Yaskawa INFORM job: DEMO_ROOF_SIDE_0625_3PAINT_7.JBI

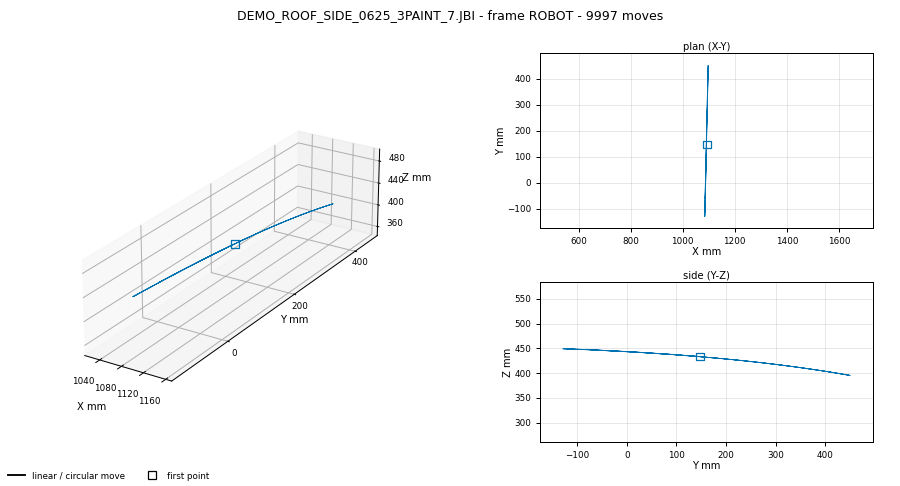
[picture p0: tool path of DEMO_ROOF_SIDE_0625_3PAINT_7.JBI in frame ROBOT, 9997 of 9997 moves have a stored position in this frame; points joined in program order, loops and branches not executed]
/JOB
//NAME DEMO_ROOF_SIDE_0625_3PAINT7
//POS
///NPOS 9997,0,0,0,0,0
///TOOL 0
///USER 0
///POSTYPE ROBOT
///RECTAN
///RCONF 1,0,0,0,0,0,0,0,0,0,0,0,0,0,0,0,0,0,0,0,0,0,0,0
C00000=1091.949,146.873,433.613,176.047,18.717,152.771
C00001=1091.943,146.623,433.633,176.045,18.716,152.771
C00002=1091.938,146.374,433.654,176.043,18.715,152.771
C00003=1091.932,146.126,433.675,176.040,18.714,152.771
C00004=1091.926,145.877,433.695,176.037,18.713,152.772
C00005=1091.921,145.628,433.716,176.034,18.712,152.772
C00006=1091.914,145.378,433.736,176.032,18.711,152.772
C00007=1091.909,145.129,433.757,176.029,18.710,152.772
C00008=1091.904,144.880,433.777,176.027,18.709,152.773
C00009=1091.899,144.631,433.798,176.024,18.708,152.773
C00010=1091.893,144.382,433.818,176.021,18.707,152.773
C00011=1091.886,144.106,433.841,176.018,18.706,152.773
C00012=1091.881,143.828,433.863,176.016,18.705,152.774
C00013=1091.874,143.552,433.886,176.013,18.704,152.774
C00014=1091.868,143.275,433.908,176.010,18.703,152.774
C00015=1091.862,143.026,433.929,176.007,18.702,152.775
C00016=1091.857,142.777,433.950,176.004,18.701,152.775
C00017=1091.851,142.527,433.970,176.002,18.700,152.775
C00018=1091.845,142.278,433.990,176.000,18.699,152.775
C00019=1091.839,142.029,434.010,175.997,18.698,152.776
C00020=1091.834,141.780,434.031,175.994,18.697,152.776
C00021=1091.829,141.531,434.051,175.991,18.696,152.776
C00022=1091.823,141.282,434.071,175.990,18.695,152.776
C00023=1091.818,141.033,434.092,175.987,18.694,152.777
C00024=1091.812,140.784,434.113,175.984,18.693,152.777
C00025=1091.806,140.535,434.133,175.981,18.692,152.777
C00026=1091.801,140.286,434.153,175.979,18.691,152.778
C00027=1091.795,140.036,434.173,175.977,18.690,152.778
C00028=1091.790,139.787,434.193,175.974,18.689,152.778
C00029=1091.784,139.538,434.213,175.971,18.688,152.778
C00030=1091.778,139.289,434.234,175.969,18.687,152.778
C00031=1091.772,139.040,434.254,175.967,18.686,152.779
C00032=1091.767,138.791,434.274,175.964,18.685,152.779
C00033=1091.761,138.542,434.293,175.961,18.683,152.779
C00034=1091.756,138.292,434.314,175.958,18.682,152.779
C00035=1091.750,138.044,434.334,175.957,18.682,152.780
C00036=1091.745,137.795,434.355,175.954,18.681,152.780
C00037=1091.739,137.546,434.375,175.951,18.679,152.780
C00038=1091.734,137.296,434.394,175.948,18.678,152.781
C00039=1091.728,137.047,434.414,175.946,18.678,152.781
C00040=1091.723,136.798,434.435,175.944,18.677,152.781
C00041=1091.717,136.549,434.455,175.941,18.676,152.781
C00042=1091.711,136.300,434.474,175.938,18.674,152.782
C00043=1091.706,136.051,434.495,175.936,18.674,152.782
C00044=1091.699,135.801,434.515,175.934,18.672,152.782
C00045=1091.694,135.552,434.536,175.931,18.671,152.782
C00046=1091.688,135.303,434.555,175.928,18.670,152.782
C00047=1091.682,135.054,434.575,175.926,18.669,152.783
C00048=1091.677,134.805,434.595,175.924,18.668,152.783
C00049=1091.671,134.555,434.615,175.921,18.667,152.783
C00050=1091.666,134.306,434.635,175.918,18.666,152.783
C00051=1091.661,134.058,434.655,175.916,18.665,152.784
C00052=1091.655,133.809,434.674,175.914,18.664,152.784
C00053=1091.650,133.559,434.694,175.911,18.663,152.784
C00054=1091.644,133.310,434.714,175.908,18.662,152.784
C00055=1091.638,133.061,434.734,175.906,18.661,152.785
C00056=1091.633,132.812,434.754,175.903,18.660,152.785
C00057=1091.627,132.563,434.773,175.901,18.658,152.785
C00058=1091.622,132.314,434.794,175.898,18.657,152.785
C00059=1091.616,132.064,434.813,175.896,18.657,152.785
C00060=1091.610,131.815,434.833,175.894,18.656,152.786
C00061=1091.604,131.566,434.853,175.891,18.655,152.786
C00062=1091.598,131.317,434.872,175.889,18.654,152.786
C00063=1091.593,131.068,434.893,175.886,18.652,152.786
C00064=1091.587,130.818,434.912,175.884,18.651,152.787
C00065=1091.581,130.570,434.932,175.881,18.650,152.787
C00066=1091.576,130.320,434.951,175.879,18.650,152.787
C00067=1091.570,130.071,434.971,175.876,18.648,152.787
C00068=1091.564,129.822,434.991,175.873,18.647,152.788
C00069=1091.559,129.573,435.011,175.871,18.646,152.788
C00070=1091.553,129.323,435.030,175.869,18.645,152.788
C00071=1091.547,129.075,435.050,175.866,18.644,152.788
C00072=1091.541,128.825,435.070,175.864,18.643,152.789
C00073=1091.536,128.576,435.089,175.862,18.642,152.789
C00074=1091.530,128.327,435.109,175.859,18.641,152.789
C00075=1091.524,128.050,435.131,175.856,18.640,152.789
C00076=1091.518,127.773,435.152,175.854,18.639,152.789
C00077=1091.511,127.496,435.174,175.851,18.637,152.790
C00078=1091.505,127.220,435.196,175.848,18.636,152.790
C00079=1091.499,126.970,435.215,175.845,18.635,152.790
C00080=1091.493,126.721,435.235,175.843,18.634,152.790
C00081=1091.488,126.472,435.254,175.841,18.633,152.791
C00082=1091.482,126.222,435.273,175.838,18.632,152.791
C00083=1091.477,125.974,435.294,175.836,18.630,152.791
C00084=1091.472,125.725,435.313,175.833,18.629,152.791
C00085=1091.466,125.475,435.332,175.831,18.629,152.792
C00086=1091.460,125.226,435.352,175.829,18.627,152.792
C00087=1091.454,124.977,435.371,175.826,18.626,152.792
C00088=1091.448,124.727,435.391,175.824,18.625,152.792
C00089=1091.442,124.479,435.411,175.821,18.624,152.792
C00090=1091.437,124.230,435.429,175.819,18.623,152.793
C00091=1091.432,123.980,435.449,175.817,18.622,152.793
C00092=1091.426,123.731,435.468,175.814,18.620,152.793
C00093=1091.420,123.482,435.488,175.811,18.619,152.793
C00094=1091.414,123.233,435.507,175.809,18.618,152.793
C00095=1091.409,122.983,435.526,175.807,18.617,152.794
C00096=1091.404,122.735,435.545,175.804,18.616,152.794
C00097=1091.398,122.485,435.564,175.802,18.615,152.794
C00098=1091.392,122.236,435.584,175.800,18.614,152.794
C00099=1091.386,121.987,435.604,175.797,18.613,152.794
C00100=1091.381,121.737,435.623,175.795,18.611,152.795
C00101=1091.376,121.488,435.642,175.793,18.611,152.795
C00102=1091.370,121.239,435.662,175.790,18.609,152.795
C00103=1091.365,120.990,435.681,175.787,18.608,152.795
C00104=1091.359,120.741,435.701,175.786,18.607,152.795
C00105=1091.353,120.491,435.720,175.783,18.606,152.796
C00106=1091.348,120.243,435.739,175.780,18.605,152.796
C00107=1091.342,119.993,435.758,175.778,18.603,152.796
C00108=1091.337,119.744,435.777,175.776,18.602,152.796
C00109=1091.331,119.494,435.797,175.773,18.601,152.796
C00110=1091.326,119.246,435.816,175.771,18.600,152.797
C00111=1091.320,118.996,435.835,175.769,18.599,152.797
C00112=1091.314,118.747,435.853,175.766,18.598,152.797
C00113=1091.309,118.498,435.872,175.764,18.596,152.797
C00114=1091.303,118.249,435.892,175.762,18.595,152.797
C00115=1091.297,117.999,435.911,175.759,18.594,152.797
C00116=1091.292,117.750,435.930,175.757,18.593,152.798
C00117=1091.287,117.501,435.949,175.755,18.592,152.798
C00118=1091.281,117.252,435.968,175.752,18.590,152.798
C00119=1091.275,117.002,435.987,175.750,18.589,152.798
C00120=1091.270,116.754,436.006,175.748,18.588,152.798
C00121=1091.264,116.504,436.026,175.745,18.587,152.798
C00122=1091.259,116.255,436.045,175.743,18.585,152.799
C00123=1091.254,116.006,436.064,175.741,18.585,152.799
C00124=1091.248,115.757,436.083,175.738,18.583,152.799
C00125=1091.242,115.507,436.102,175.736,18.581,152.799
C00126=1091.237,115.258,436.121,175.734,18.581,152.799
C00127=1091.231,115.009,436.140,175.731,18.579,152.799
C00128=1091.226,114.760,436.160,175.729,18.578,152.800
C00129=1091.220,114.511,436.178,175.726,18.577,152.800
C00130=1091.214,114.262,436.197,175.724,18.575,152.800
C00131=1091.209,114.012,436.216,175.722,18.574,152.800
C00132=1091.204,113.763,436.234,175.720,18.573,152.800
C00133=1091.198,113.514,436.254,175.717,18.572,152.801
C00134=1091.192,113.264,436.272,175.715,18.571,152.801
C00135=1091.187,113.016,436.291,175.713,18.570,152.801
C00136=1091.181,112.766,436.310,175.710,18.568,152.801
C00137=1091.175,112.517,436.330,175.708,18.567,152.801
C00138=1091.170,112.268,436.347,175.706,18.566,152.801
C00139=1091.164,111.990,436.369,175.703,18.565,152.802
C00140=1091.157,111.714,436.390,175.701,18.564,152.802
C00141=1091.151,111.437,436.411,175.698,18.562,152.802
C00142=1091.145,111.160,436.431,175.695,18.561,152.802
C00143=1091.139,110.911,436.451,175.693,18.559,152.802
C00144=1091.133,110.661,436.468,175.690,18.558,152.802
C00145=1091.128,110.413,436.487,175.689,18.557,152.803
C00146=1091.122,110.163,436.507,175.686,18.555,152.803
C00147=1091.116,109.915,436.525,175.684,18.555,152.803
C00148=1091.111,109.665,436.543,175.682,18.553,152.803
C00149=1091.104,109.416,436.562,175.679,18.552,152.803
C00150=1091.099,109.167,436.581,175.677,18.551,152.804
C00151=1091.094,108.917,436.599,175.675,18.550,152.804
C00152=1091.087,108.668,436.618,175.672,18.548,152.804
C00153=1091.082,108.419,436.637,175.670,18.547,152.804
C00154=1091.076,108.169,436.655,175.668,18.546,152.804
C00155=1091.071,107.920,436.674,175.665,18.545,152.804
C00156=1091.065,107.671,436.693,175.663,18.544,152.805
C00157=1091.059,107.421,436.711,175.661,18.542,152.805
C00158=1091.054,107.173,436.730,175.658,18.540,152.805
C00159=1091.048,106.923,436.748,175.657,18.540,152.805
C00160=1091.043,106.674,436.767,175.654,18.538,152.805
C00161=1091.037,106.425,436.785,175.652,18.537,152.805
C00162=1091.031,106.175,436.804,175.650,18.536,152.806
C00163=1091.026,105.926,436.823,175.647,18.534,152.806
C00164=1091.020,105.677,436.841,175.645,18.533,152.806
C00165=1091.015,105.428,436.859,175.643,18.532,152.806
C00166=1091.008,105.179,436.878,175.640,18.531,152.806
C00167=1091.004,104.929,436.896,175.639,18.530,152.806
C00168=1090.997,104.680,436.915,175.636,18.528,152.806
C00169=1090.993,104.431,436.933,175.634,18.527,152.806
C00170=1090.986,104.182,436.952,175.632,18.526,152.807
C00171=1090.981,103.932,436.970,175.629,18.524,152.807
C00172=1090.975,103.683,436.989,175.627,18.523,152.807
C00173=1090.970,103.434,437.007,175.625,18.522,152.807
C00174=1090.964,103.185,437.025,175.622,18.521,152.807
C00175=1090.959,102.935,437.044,175.621,18.519,152.807
C00176=1090.952,102.686,437.062,175.618,18.518,152.808
C00177=1090.948,102.437,437.080,175.616,18.517,152.808
C00178=1090.942,102.187,437.098,175.614,18.515,152.808
C00179=1090.936,101.938,437.117,175.611,18.514,152.808
C00180=1090.930,101.689,437.135,175.609,18.513,152.808
C00181=1090.925,101.440,437.154,175.607,18.511,152.808
C00182=1090.919,101.190,437.172,175.604,18.510,152.808
C00183=1090.914,100.941,437.191,175.603,18.509,152.808
C00184=1090.908,100.692,437.209,175.600,18.507,152.809
C00185=1090.902,100.443,437.226,175.598,18.507,152.809
C00186=1090.897,100.193,437.246,175.596,18.505,152.809
C00187=1090.891,99.944,437.263,175.593,18.503,152.809
C00188=1090.885,99.694,437.281,175.592,18.502,152.809
C00189=1090.880,99.446,437.300,175.589,18.501,152.809
C00190=1090.874,99.196,437.318,175.587,18.500,152.810
C00191=1090.868,98.947,437.335,175.585,18.499,152.810
C00192=1090.863,98.697,437.355,175.582,18.497,152.810
C00193=1090.857,98.448,437.372,175.581,18.496,152.810
C00194=1090.851,98.199,437.390,175.578,18.494,152.810
C00195=1090.845,97.950,437.408,175.577,18.493,152.810
C00196=1090.840,97.700,437.427,175.574,18.492,152.810
C00197=1090.834,97.451,437.445,175.571,18.491,152.811
C00198=1090.828,97.201,437.462,175.570,18.489,152.811
C00199=1090.823,96.953,437.481,175.567,18.488,152.811
C00200=1090.817,96.703,437.499,175.565,18.487,152.811
C00201=1090.811,96.454,437.517,175.563,18.485,152.811
C00202=1090.806,96.205,437.534,175.560,18.484,152.811
C00203=1090.800,95.928,437.555,175.559,18.483,152.811
C00204=1090.793,95.650,437.575,175.556,18.481,152.811
C00205=1090.787,95.374,437.595,175.554,18.479,152.811
C00206=1090.781,95.098,437.615,175.551,18.478,152.812
C00207=1090.775,94.849,437.633,175.549,18.477,152.812
C00208=1090.770,94.599,437.651,175.547,18.476,152.812
C00209=1090.764,94.350,437.669,175.544,18.474,152.812
C00210=1090.759,94.100,437.687,175.543,18.473,152.812
C00211=1090.752,93.851,437.705,175.540,18.471,152.812
C00212=1090.747,93.602,437.722,175.538,18.470,152.812
C00213=1090.742,93.353,437.741,175.536,18.469,152.812
C00214=1090.736,93.103,437.759,175.534,18.467,152.813
C00215=1090.730,92.854,437.777,175.532,18.466,152.813
C00216=1090.725,92.605,437.794,175.529,18.464,152.813
C00217=1090.719,92.355,437.813,175.527,18.463,152.813
C00218=1090.714,92.106,437.830,175.525,18.462,152.813
C00219=1090.708,91.857,437.848,175.523,18.460,152.813
C00220=1090.702,91.607,437.866,175.521,18.459,152.813
C00221=1090.697,91.358,437.883,175.519,18.458,152.813
C00222=1090.692,91.109,437.901,175.517,18.456,152.814
C00223=1090.686,90.859,437.919,175.514,18.455,152.814
C00224=1090.680,90.610,437.937,175.512,18.453,152.814
C00225=1090.674,90.360,437.955,175.510,18.452,152.814
C00226=1090.669,90.111,437.972,175.508,18.451,152.814
C00227=1090.663,89.862,437.990,175.506,18.450,152.814
C00228=1090.657,89.613,438.008,175.504,18.448,152.814
C00229=1090.651,89.363,438.025,175.502,18.447,152.814
C00230=1090.646,89.114,438.043,175.499,18.445,152.814
C00231=1090.640,88.865,438.061,175.497,18.444,152.815
C00232=1090.634,88.616,438.079,175.495,18.443,152.815
C00233=1090.629,88.367,438.096,175.493,18.441,152.815
C00234=1090.623,88.117,438.114,175.491,18.440,152.815
C00235=1090.617,87.868,438.132,175.489,18.438,152.815
C00236=1090.612,87.619,438.149,175.487,18.437,152.815
C00237=1090.605,87.369,438.167,175.485,18.436,152.815
C00238=1090.600,87.120,438.185,175.482,18.434,152.815
C00239=1090.594,86.871,438.202,175.480,18.433,152.815
C00240=1090.589,86.621,438.219,175.478,18.431,152.816
C00241=1090.583,86.372,438.237,175.476,18.430,152.816
C00242=1090.578,86.123,438.255,175.474,18.429,152.816
C00243=1090.571,85.873,438.273,175.472,18.427,152.816
C00244=1090.566,85.624,438.290,175.470,18.426,152.816
C00245=1090.560,85.375,438.308,175.468,18.425,152.816
C00246=1090.554,85.126,438.325,175.466,18.423,152.816
C00247=1090.548,84.876,438.342,175.463,18.421,152.816
C00248=1090.543,84.627,438.359,175.461,18.420,152.816
C00249=1090.537,84.378,438.377,175.459,18.419,152.816
C00250=1090.532,84.129,438.395,175.457,18.418,152.817
C00251=1090.526,83.879,438.412,175.455,18.416,152.817
C00252=1090.520,83.629,438.429,175.453,18.414,152.817
C00253=1090.515,83.380,438.447,175.451,18.413,152.817
C00254=1090.509,83.131,438.464,175.449,18.412,152.817
C00255=1090.503,82.881,438.482,175.447,18.410,152.817
C00256=1090.498,82.632,438.499,175.444,18.409,152.817
C00257=1090.493,82.383,438.517,175.443,18.408,152.817
C00258=1090.487,82.134,438.534,175.440,18.406,152.817
C00259=1090.482,81.884,438.551,175.439,18.404,152.817
C00260=1090.475,81.634,438.569,175.436,18.403,152.817
C00261=1090.469,81.385,438.586,175.435,18.402,152.817
C00262=1090.464,81.136,438.604,175.432,18.400,152.818
C00263=1090.459,80.887,438.621,175.430,18.399,152.818
C00264=1090.453,80.638,438.638,175.428,18.397,152.818
C00265=1090.448,80.389,438.656,175.427,18.396,152.818
C00266=1090.442,80.138,438.673,175.424,18.394,152.818
C00267=1090.436,79.862,438.692,175.422,18.393,152.818
C00268=1090.429,79.585,438.711,175.419,18.391,152.818
C00269=1090.423,79.308,438.730,175.418,18.390,152.818
C00270=1090.416,79.032,438.749,175.415,18.388,152.818
C00271=1090.411,78.782,438.767,175.413,18.386,152.818
C00272=1090.406,78.533,438.784,175.411,18.385,152.818
C00273=1090.400,78.284,438.801,175.409,18.383,152.818
C00274=1090.395,78.034,438.818,175.407,18.382,152.819
C00275=1090.389,77.785,438.835,175.405,18.381,152.819
C00276=1090.383,77.536,438.853,175.403,18.379,152.819
C00277=1090.377,77.286,438.870,175.401,18.377,152.819
C00278=1090.371,77.037,438.887,175.399,18.376,152.819
C00279=1090.366,76.788,438.904,175.397,18.375,152.819
C00280=1090.360,76.539,438.921,175.394,18.373,152.819
C00281=1090.355,76.289,438.938,175.392,18.372,152.819
C00282=1090.348,76.039,438.955,175.390,18.370,152.819
C00283=1090.343,75.790,438.972,175.388,18.369,152.819
C00284=1090.338,75.541,438.990,175.386,18.367,152.819
C00285=1090.332,75.291,439.006,175.384,18.366,152.820
C00286=1090.326,75.042,439.024,175.382,18.364,152.820
C00287=1090.321,74.793,439.041,175.380,18.363,152.820
C00288=1090.315,74.544,439.057,175.378,18.362,152.820
C00289=1090.309,74.294,439.074,175.377,18.360,152.820
C00290=1090.303,74.045,439.092,175.374,18.358,152.820
C00291=1090.297,73.795,439.109,175.372,18.357,152.820
C00292=1090.292,73.546,439.125,175.370,18.356,152.820
C00293=1090.286,73.297,439.142,175.368,18.354,152.820
C00294=1090.281,73.047,439.159,175.366,18.353,152.820
C00295=1090.275,72.798,439.177,175.364,18.351,152.820
C00296=1090.269,72.549,439.193,175.362,18.349,152.820
C00297=1090.264,72.299,439.210,175.360,18.348,152.820
C00298=1090.258,72.050,439.227,175.358,18.347,152.820
C00299=1090.252,71.801,439.244,175.357,18.345,152.820
C00300=1090.247,71.551,439.261,175.354,18.344,152.821
C00301=1090.240,71.302,439.278,175.352,18.342,152.821
C00302=1090.235,71.052,439.295,175.350,18.340,152.821
C00303=1090.230,70.802,439.312,175.348,18.339,152.821
C00304=1090.224,70.554,439.329,175.346,18.338,152.821
C00305=1090.219,70.304,439.345,175.345,18.336,152.821
C00306=1090.213,70.055,439.362,175.342,18.335,152.821
C00307=1090.207,69.806,439.379,175.340,18.333,152.821
C00308=1090.201,69.556,439.395,175.338,18.331,152.821
C00309=1090.196,69.307,439.412,175.337,18.330,152.821
C00310=1090.190,69.058,439.429,175.334,18.329,152.821
C00311=1090.184,68.808,439.446,175.333,18.327,152.821
C00312=1090.178,68.559,439.462,175.330,18.326,152.821
C00313=1090.173,68.309,439.479,175.328,18.325,152.821
C00314=1090.167,68.060,439.496,175.326,18.322,152.821
C00315=1090.162,67.811,439.513,175.325,18.321,152.821
C00316=1090.156,67.561,439.529,175.322,18.319,152.821
C00317=1090.151,67.312,439.546,175.321,18.318,152.822
C00318=1090.145,67.062,439.562,175.318,18.317,152.822
C00319=1090.138,66.814,439.579,175.317,18.315,152.822
C00320=1090.133,66.564,439.596,175.314,18.313,152.822
C00321=1090.127,66.315,439.613,175.313,18.312,152.822
C00322=1090.122,66.065,439.629,175.310,18.310,152.822
C00323=1090.116,65.816,439.646,175.309,18.309,152.822
C00324=1090.111,65.566,439.662,175.307,18.307,152.822
C00325=1090.105,65.317,439.679,175.305,18.306,152.822
C00326=1090.099,65.068,439.696,175.303,18.304,152.822
C00327=1090.093,64.818,439.713,175.301,18.303,152.822
C00328=1090.088,64.569,439.729,175.298,18.301,152.822
C00329=1090.082,64.319,439.746,175.297,18.300,152.822
C00330=1090.076,64.070,439.762,175.295,18.298,152.822
C00331=1090.069,63.793,439.781,175.293,18.297,152.822
C00332=1090.063,63.516,439.799,175.291,18.295,152.822
C00333=1090.057,63.239,439.816,175.288,18.293,152.823
C00334=1090.050,62.963,439.836,175.286,18.291,152.823
C00335=1090.044,62.713,439.852,175.284,18.290,152.823
C00336=1090.038,62.464,439.868,175.282,18.289,152.823
C00337=1090.032,62.215,439.884,175.280,18.287,152.823
C00338=1090.027,61.965,439.901,175.278,18.285,152.823
C00339=1090.021,61.716,439.918,175.277,18.284,152.823
C00340=1090.015,61.466,439.934,175.274,18.282,152.823
C00341=1090.009,61.217,439.950,175.272,18.281,152.823
C00342=1090.004,60.967,439.967,175.271,18.280,152.823
C00343=1089.998,60.718,439.983,175.268,18.278,152.823
C00344=1089.992,60.468,439.999,175.267,18.276,152.823
C00345=1089.986,60.219,440.016,175.265,18.275,152.823
C00346=1089.980,59.970,440.032,175.263,18.273,152.823
C00347=1089.975,59.721,440.048,175.261,18.272,152.823
C00348=1089.969,59.471,440.065,175.259,18.271,152.823
C00349=1089.964,59.222,440.081,175.257,18.269,152.823
C00350=1089.958,58.973,440.097,175.255,18.268,152.823
C00351=1089.952,58.723,440.113,175.253,18.265,152.823
C00352=1089.946,58.473,440.129,175.251,18.264,152.824
C00353=1089.941,58.224,440.146,175.249,18.262,152.824
C00354=1089.935,57.974,440.162,175.247,18.261,152.824
C00355=1089.929,57.725,440.178,175.245,18.259,152.824
C00356=1089.923,57.476,440.195,175.243,18.258,152.824
C00357=1089.917,57.226,440.211,175.242,18.256,152.824
C00358=1089.911,56.977,440.227,175.240,18.255,152.824
C00359=1089.905,56.728,440.243,175.238,18.253,152.824
C00360=1089.901,56.478,440.259,175.236,18.252,152.824
C00361=1089.895,56.229,440.275,175.234,18.250,152.824
C00362=1089.889,55.979,440.292,175.232,18.249,152.824
C00363=1089.883,55.730,440.308,175.230,18.247,152.824
C00364=1089.877,55.481,440.324,175.228,18.245,152.824
C00365=1089.871,55.231,440.340,175.226,18.244,152.824
C00366=1089.865,54.981,440.356,175.224,18.242,152.824
C00367=1089.859,54.732,440.372,175.223,18.241,152.824
C00368=1089.855,54.483,440.389,175.221,18.240,152.824
C00369=1089.849,54.234,440.405,175.219,18.237,152.824
C00370=1089.843,53.984,440.420,175.217,18.236,152.824
C00371=1089.837,53.734,440.437,175.215,18.234,152.824
C00372=1089.831,53.485,440.453,175.213,18.233,152.824
C00373=1089.825,53.236,440.469,175.211,18.231,152.824
C00374=1089.820,52.986,440.484,175.210,18.230,152.824
C00375=1089.814,52.737,440.501,175.207,18.228,152.824
C00376=1089.808,52.488,440.517,175.206,18.226,152.824
C00377=1089.802,52.238,440.533,175.204,18.225,152.824
C00378=1089.797,51.988,440.549,175.202,18.223,152.824
C00379=1089.791,51.740,440.565,175.200,18.222,152.824
C00380=1089.786,51.490,440.581,175.198,18.220,152.825
C00381=1089.781,51.240,440.597,175.196,18.219,152.824
C00382=1089.775,50.991,440.613,175.194,18.216,152.824
C00383=1089.769,50.741,440.630,175.193,18.215,152.825
C00384=1089.764,50.492,440.645,175.190,18.213,152.825
C00385=1089.758,50.243,440.661,175.189,18.212,152.824
C00386=1089.752,49.993,440.677,175.187,18.211,152.825
C00387=1089.746,49.744,440.693,175.185,18.209,152.825
C00388=1089.741,49.495,440.709,175.184,18.207,152.825
C00389=1089.735,49.245,440.724,175.181,18.205,152.825
C00390=1089.729,48.996,440.740,175.180,18.204,152.825
C00391=1089.724,48.746,440.756,175.178,18.202,152.825
C00392=1089.718,48.497,440.772,175.176,18.201,152.825
C00393=1089.712,48.248,440.788,175.174,18.199,152.825
C00394=1089.707,47.998,440.804,175.172,18.197,152.825
C00395=1089.700,47.721,440.821,175.170,18.195,152.825
C00396=1089.694,47.443,440.839,175.168,18.194,152.825
C00397=1089.688,47.167,440.856,175.166,18.192,152.825
C00398=1089.682,46.890,440.874,175.164,18.190,152.825
C00399=1089.676,46.640,440.889,175.162,18.189,152.825
C00400=1089.670,46.391,440.906,175.160,18.186,152.825
C00401=1089.665,46.142,440.921,175.159,18.185,152.825
C00402=1089.659,45.892,440.937,175.157,18.184,152.825
C00403=1089.653,45.642,440.953,175.155,18.182,152.825
C00404=1089.648,45.394,440.969,175.153,18.180,152.825
C00405=1089.642,45.144,440.984,175.151,18.178,152.825
C00406=1089.636,44.894,441.000,175.149,18.177,152.825
C00407=1089.631,44.645,441.016,175.147,18.175,152.825
C00408=1089.625,44.396,441.032,175.146,18.173,152.825
C00409=1089.620,44.146,441.047,175.144,18.172,152.825
C00410=1089.615,43.896,441.063,175.142,18.170,152.825
C00411=1089.609,43.647,441.079,175.141,18.169,152.825
C00412=1089.603,43.397,441.094,175.138,18.166,152.825
C00413=1089.598,43.148,441.110,175.137,18.165,152.825
C00414=1089.591,42.899,441.125,175.135,18.164,152.825
C00415=1089.586,42.649,441.141,175.133,18.162,152.825
C00416=1089.580,42.400,441.157,175.132,18.160,152.825
C00417=1089.575,42.150,441.172,175.129,18.159,152.825
C00418=1089.569,41.901,441.188,175.128,18.157,152.825
C00419=1089.562,41.651,441.203,175.126,18.155,152.825
C00420=1089.557,41.402,441.219,175.124,18.154,152.825
C00421=1089.551,41.153,441.235,175.122,18.152,152.825
C00422=1089.546,40.903,441.250,175.120,18.150,152.825
C00423=1089.540,40.654,441.265,175.119,18.149,152.825
C00424=1089.534,40.404,441.281,175.116,18.147,152.825
C00425=1089.529,40.155,441.296,175.115,18.145,152.825
C00426=1089.523,39.905,441.312,175.114,18.144,152.825
C00427=1089.517,39.655,441.327,175.111,18.142,152.825
C00428=1089.512,39.407,441.343,175.110,18.141,152.825
C00429=1089.506,39.157,441.358,175.107,18.139,152.825
C00430=1089.500,38.907,441.374,175.106,18.137,152.825
C00431=1089.495,38.658,441.388,175.104,18.136,152.825
C00432=1089.489,38.409,441.405,175.102,18.134,152.825
C00433=1089.484,38.159,441.420,175.101,18.132,152.825
C00434=1089.478,37.909,441.435,175.099,18.130,152.825
C00435=1089.472,37.660,441.450,175.097,18.129,152.825
C00436=1089.466,37.411,441.466,175.095,18.128,152.825
C00437=1089.461,37.161,441.482,175.093,18.125,152.825
C00438=1089.454,36.911,441.497,175.092,18.124,152.825
C00439=1089.449,36.662,441.512,175.090,18.123,152.825
C00440=1089.443,36.412,441.527,175.088,18.121,152.825
C00441=1089.437,36.164,441.543,175.087,18.119,152.825
C00442=1089.431,35.914,441.558,175.084,18.117,152.825
C00443=1089.425,35.664,441.573,175.083,18.116,152.825
C00444=1089.420,35.415,441.588,175.081,18.114,152.825
C00445=1089.414,35.165,441.603,175.079,18.112,152.825
C00446=1089.408,34.915,441.619,175.077,18.111,152.825
C00447=1089.402,34.667,441.634,175.075,18.109,152.825
C00448=1089.397,34.417,441.650,175.074,18.108,152.825
C00449=1089.391,34.168,441.664,175.072,18.106,152.825
C00450=1089.385,33.918,441.680,175.070,18.104,152.825
C00451=1089.380,33.669,441.695,175.068,18.103,152.825
C00452=1089.374,33.419,441.710,175.067,18.101,152.825
C00453=1089.368,33.169,441.725,175.065,18.099,152.825
C00454=1089.362,32.920,441.740,175.063,18.098,152.825
C00455=1089.357,32.670,441.756,175.061,18.096,152.825
C00456=1089.351,32.421,441.770,175.060,18.094,152.825
C00457=1089.345,32.171,441.786,175.058,18.093,152.825
C00458=1089.339,31.922,441.800,175.056,18.091,152.825
C00459=1089.333,31.646,441.818,175.055,18.089,152.825
C00460=1089.326,31.368,441.835,175.052,18.088,152.825
C00461=1089.320,31.091,441.852,175.050,18.085,152.825
C00462=1089.314,30.814,441.868,175.048,18.084,152.825
C00463=1089.309,30.565,441.883,175.046,18.082,152.825
C00464=1089.302,30.315,441.898,175.045,18.080,152.825
C00465=1089.297,30.066,441.913,175.043,18.079,152.825
C00466=1089.291,29.816,441.928,175.041,18.077,152.825
C00467=1089.286,29.567,441.943,175.040,18.075,152.825
C00468=1089.279,29.317,441.958,175.038,18.074,152.825
C00469=1089.274,29.068,441.973,175.036,18.072,152.825
C00470=1089.268,28.819,441.988,175.035,18.070,152.825
C00471=1089.263,28.569,442.004,175.032,18.068,152.825
C00472=1089.256,28.320,442.018,175.031,18.067,152.825
C00473=1089.251,28.070,442.034,175.029,18.065,152.825
C00474=1089.245,27.820,442.048,175.027,18.063,152.825
C00475=1089.240,27.571,442.062,175.026,18.062,152.825
C00476=1089.234,27.321,442.078,175.024,18.060,152.825
C00477=1089.228,27.072,442.093,175.022,18.059,152.825
C00478=1089.222,26.823,442.108,175.020,18.057,152.825
C00479=1089.217,26.573,442.123,175.019,18.055,152.825
C00480=1089.210,26.324,442.138,175.017,18.053,152.825
C00481=1089.204,26.075,442.152,175.015,18.052,152.825
C00482=1089.199,25.825,442.168,175.014,18.051,152.825
C00483=1089.193,25.575,442.182,175.011,18.049,152.825
C00484=1089.187,25.325,442.197,175.010,18.047,152.825
C00485=1089.182,25.076,442.212,175.008,18.045,152.825
C00486=1089.176,24.827,442.227,175.006,18.043,152.825
C00487=1089.170,24.578,442.241,175.005,18.042,152.825
C00488=1089.164,24.327,442.256,175.003,18.040,152.825
C00489=1089.159,24.078,442.271,175.001,18.039,152.825
C00490=1089.152,23.828,442.286,175.000,18.037,152.825
C00491=1089.147,23.579,442.301,174.998,18.035,152.825
C00492=1089.141,23.329,442.316,174.996,18.033,152.825
C00493=1089.135,23.080,442.330,174.995,18.032,152.825
C00494=1089.130,22.831,442.345,174.992,18.030,152.825
C00495=1089.124,22.581,442.360,174.991,18.029,152.825
C00496=1089.118,22.332,442.374,174.990,18.027,152.825
C00497=1089.112,22.082,442.389,174.987,18.025,152.825
C00498=1089.107,21.832,442.404,174.986,18.023,152.825
C00499=1089.101,21.584,442.418,174.985,18.022,152.825
C00500=1089.095,21.334,442.433,174.982,18.020,152.825
C00501=1089.089,21.084,442.447,174.981,18.019,152.825
C00502=1089.084,20.834,442.463,174.979,18.017,152.825
C00503=1089.078,20.585,442.477,174.977,18.015,152.825
C00504=1089.073,20.336,442.491,174.976,18.013,152.825
C00505=1089.066,20.086,442.506,174.974,18.012,152.825
C00506=1089.061,19.837,442.521,174.972,18.010,152.825
C00507=1089.055,19.587,442.535,174.971,18.008,152.825
C00508=1089.049,19.338,442.550,174.969,18.007,152.825
C00509=1089.043,19.089,442.565,174.967,18.005,152.825
C00510=1089.037,18.838,442.579,174.965,18.003,152.825
C00511=1089.032,18.589,442.593,174.964,18.002,152.825
C00512=1089.026,18.339,442.608,174.962,18.000,152.825
C00513=1089.020,18.090,442.623,174.960,17.998,152.825
C00514=1089.015,17.841,442.637,174.959,17.997,152.824
C00515=1089.009,17.591,442.652,174.957,17.994,152.824
C00516=1089.003,17.342,442.666,174.955,17.993,152.825
C00517=1088.997,17.091,442.680,174.954,17.992,152.825
C00518=1088.991,16.842,442.695,174.951,17.990,152.825
C00519=1088.986,16.593,442.710,174.950,17.988,152.824
C00520=1088.980,16.343,442.724,174.949,17.987,152.824
C00521=1088.974,16.094,442.739,174.946,17.984,152.824
C00522=1088.969,15.844,442.753,174.945,17.983,152.824
C00523=1088.962,15.569,442.769,174.944,17.981,152.824
C00524=1088.956,15.293,442.785,174.941,17.979,152.824
C00525=1088.949,15.017,442.800,174.939,17.977,152.824
C00526=1088.943,14.742,442.817,174.938,17.975,152.824
C00527=1088.937,14.492,442.831,174.936,17.974,152.824
C00528=1088.931,14.243,442.845,174.934,17.972,152.824
C00529=1088.925,13.993,442.860,174.933,17.971,152.824
C00530=1088.919,13.744,442.874,174.931,17.969,152.824
C00531=1088.914,13.494,442.888,174.929,17.967,152.824
C00532=1088.907,13.245,442.903,174.928,17.965,152.824
C00533=1088.902,12.995,442.917,174.926,17.964,152.824
C00534=1088.896,12.746,442.932,174.924,17.962,152.824
C00535=1088.890,12.496,442.946,174.922,17.961,152.824
C00536=1088.885,12.246,442.960,174.921,17.959,152.824
C00537=1088.879,11.997,442.974,174.919,17.957,152.824
C00538=1088.873,11.747,442.988,174.917,17.955,152.824
C00539=1088.867,11.498,443.003,174.916,17.954,152.824
C00540=1088.862,11.249,443.017,174.915,17.952,152.824
C00541=1088.854,10.999,443.031,174.912,17.951,152.824
C00542=1088.849,10.750,443.045,174.911,17.949,152.824
C00543=1088.843,10.500,443.059,174.909,17.948,152.824
C00544=1088.837,10.250,443.074,174.907,17.945,152.824
C00545=1088.832,10.001,443.088,174.906,17.944,152.824
C00546=1088.826,9.751,443.102,174.904,17.942,152.824
C00547=1088.820,9.502,443.117,174.902,17.940,152.824
C00548=1088.814,9.252,443.130,174.900,17.939,152.824
C00549=1088.809,9.002,443.144,174.899,17.938,152.824
C00550=1088.803,8.754,443.159,174.898,17.936,152.824
C00551=1088.796,8.504,443.173,174.895,17.934,152.824
C00552=1088.791,8.254,443.186,174.894,17.932,152.824
C00553=1088.785,8.005,443.201,174.893,17.931,152.824
C00554=1088.779,7.755,443.215,174.890,17.929,152.824
C00555=1088.773,7.505,443.229,174.889,17.927,152.824
C00556=1088.768,7.256,443.244,174.888,17.925,152.824
C00557=1088.762,7.007,443.257,174.886,17.924,152.824
C00558=1088.757,6.757,443.271,174.884,17.922,152.824
C00559=1088.750,6.507,443.285,174.882,17.921,152.824
C00560=1088.744,6.258,443.300,174.881,17.919,152.824
C00561=1088.739,6.009,443.313,174.879,17.917,152.824
C00562=1088.733,5.759,443.327,174.877,17.915,152.824
C00563=1088.727,5.509,443.342,174.876,17.914,152.824
C00564=1088.722,5.259,443.355,174.875,17.912,152.824
C00565=1088.715,5.011,443.369,174.872,17.910,152.824
C00566=1088.710,4.761,443.383,174.871,17.909,152.824
C00567=1088.704,4.511,443.397,174.870,17.907,152.824
C00568=1088.698,4.261,443.411,174.867,17.905,152.824
C00569=1088.693,4.012,443.425,174.866,17.904,152.824
C00570=1088.687,3.763,443.440,174.864,17.902,152.824
C00571=1088.681,3.513,443.453,174.863,17.901,152.824
C00572=1088.675,3.264,443.467,174.861,17.899,152.824
C00573=1088.669,3.013,443.481,174.859,17.897,152.824
C00574=1088.664,2.764,443.495,174.858,17.895,152.823
C00575=1088.658,2.514,443.509,174.856,17.893,152.823
C00576=1088.652,2.265,443.522,174.854,17.892,152.823
C00577=1088.646,2.016,443.537,174.853,17.890,152.823
C00578=1088.641,1.767,443.551,174.852,17.889,152.823
C00579=1088.634,1.516,443.565,174.849,17.886,152.823
C00580=1088.629,1.267,443.579,174.848,17.885,152.823
C00581=1088.623,1.017,443.592,174.847,17.883,152.823
C00582=1088.617,0.768,443.606,174.845,17.882,152.823
C00583=1088.612,0.518,443.620,174.843,17.880,152.823
C00584=1088.606,0.269,443.634,174.842,17.878,152.823
C00585=1088.601,0.019,443.647,174.840,17.877,152.823
C00586=1088.595,-0.230,443.661,174.838,17.875,152.823
C00587=1088.589,-0.504,443.676,174.836,17.873,152.823
C00588=1088.582,-0.778,443.691,174.835,17.871,152.823
C00589=1088.575,-1.052,443.706,174.833,17.869,152.823
C00590=1088.569,-1.325,443.721,174.832,17.867,152.823
C00591=1088.564,-1.575,443.735,174.829,17.865,152.823
C00592=1088.558,-1.825,443.749,174.828,17.864,152.823
C00593=1088.552,-2.074,443.762,174.827,17.862,152.823
C00594=1088.547,-2.323,443.776,174.824,17.860,152.823
C00595=1088.541,-2.573,443.790,174.823,17.859,152.823
C00596=1088.536,-2.822,443.804,174.821,17.857,152.823
C00597=1088.529,-3.072,443.817,174.820,17.856,152.823
C00598=1088.524,-3.321,443.831,174.818,17.854,152.823
C00599=1088.518,-3.571,443.845,174.816,17.852,152.823
C00600=1088.512,-3.821,443.859,174.815,17.851,152.823
C00601=1088.506,-4.070,443.872,174.814,17.849,152.823
C00602=1088.500,-4.320,443.886,174.811,17.847,152.823
C00603=1088.494,-4.569,443.900,174.810,17.845,152.823
C00604=1088.488,-4.819,443.913,174.809,17.844,152.823
C00605=1088.483,-5.068,443.927,174.807,17.842,152.823
C00606=1088.477,-5.317,443.940,174.805,17.841,152.823
C00607=1088.471,-5.567,443.954,174.803,17.839,152.823
C00608=1088.465,-5.817,443.966,174.802,17.837,152.823
C00609=1088.459,-6.067,443.981,174.800,17.836,152.823
C00610=1088.453,-6.316,443.994,174.798,17.834,152.823
C00611=1088.447,-6.566,444.008,174.797,17.832,152.823
C00612=1088.441,-6.815,444.021,174.796,17.831,152.822
C00613=1088.436,-7.065,444.035,174.794,17.829,152.822
C00614=1088.429,-7.314,444.048,174.793,17.827,152.822
C00615=1088.424,-7.564,444.061,174.790,17.826,152.823
C00616=1088.418,-7.814,444.075,174.789,17.824,152.822
C00617=1088.413,-8.063,444.088,174.787,17.823,152.822
C00618=1088.406,-8.312,444.102,174.786,17.821,152.822
C00619=1088.401,-8.562,444.116,174.784,17.819,152.822
C00620=1088.395,-8.811,444.129,174.782,17.817,152.822
C00621=1088.390,-9.061,444.142,174.781,17.816,152.822
C00622=1088.383,-9.311,444.156,174.780,17.814,152.822
C00623=1088.377,-9.561,444.169,174.777,17.812,152.822
C00624=1088.371,-9.810,444.183,174.776,17.811,152.822
C00625=1088.366,-10.060,444.196,174.775,17.809,152.822
C00626=1088.360,-10.310,444.209,174.773,17.808,152.822
C00627=1088.353,-10.559,444.222,174.771,17.806,152.822
C00628=1088.348,-10.809,444.236,174.769,17.804,152.822
C00629=1088.342,-11.058,444.249,174.768,17.803,152.822
C00630=1088.337,-11.308,444.263,174.767,17.801,152.822
C00631=1088.330,-11.557,444.276,174.765,17.799,152.822
C00632=1088.325,-11.807,444.289,174.763,17.797,152.822
C00633=1088.319,-12.057,444.302,174.762,17.796,152.822
C00634=1088.314,-12.306,444.316,174.760,17.794,152.822
C00635=1088.307,-12.556,444.329,174.759,17.793,152.822
C00636=1088.301,-12.805,444.342,174.757,17.790,152.822
C00637=1088.296,-13.055,444.356,174.755,17.789,152.822
C00638=1088.290,-13.304,444.369,174.754,17.787,152.822
C00639=1088.285,-13.554,444.382,174.752,17.786,152.822
C00640=1088.278,-13.804,444.396,174.751,17.785,152.822
C00641=1088.272,-14.054,444.408,174.749,17.783,152.822
C00642=1088.268,-14.302,444.422,174.747,17.781,152.822
C00643=1088.261,-14.552,444.435,174.746,17.779,152.822
C00644=1088.256,-14.802,444.448,174.745,17.778,152.822
C00645=1088.250,-15.051,444.461,174.742,17.776,152.822
C00646=1088.244,-15.300,444.475,174.741,17.774,152.822
C00647=1088.239,-15.551,444.488,174.740,17.773,152.822
C00648=1088.232,-15.800,444.501,174.738,17.771,152.822
C00649=1088.226,-16.050,444.514,174.737,17.770,152.822
C00650=1088.220,-16.299,444.527,174.734,17.768,152.822
C00651=1088.214,-16.572,444.541,174.733,17.766,152.822
C00652=1088.207,-16.843,444.555,174.732,17.765,152.822
C00653=1088.201,-17.115,444.569,174.729,17.762,152.822
C00654=1088.195,-17.387,444.584,174.728,17.761,152.822
C00655=1088.189,-17.637,444.598,174.727,17.759,152.822
C00656=1088.183,-17.887,444.610,174.724,17.757,152.822
C00657=1088.176,-18.136,444.623,174.723,17.756,152.821
C00658=1088.171,-18.386,444.637,174.722,17.754,152.821
C00659=1088.165,-18.635,444.650,174.720,17.753,152.822
C00660=1088.159,-18.885,444.662,174.719,17.751,152.822
C00661=1088.153,-19.134,444.676,174.716,17.749,152.822
C00662=1088.148,-19.384,444.688,174.715,17.748,152.821
C00663=1088.142,-19.633,444.702,174.714,17.746,152.821
C00664=1088.136,-19.883,444.714,174.712,17.745,152.821
C00665=1088.130,-20.132,444.728,174.711,17.743,152.821
C00666=1088.124,-20.382,444.740,174.708,17.741,152.821
C00667=1088.118,-20.632,444.753,174.707,17.740,152.821
C00668=1088.112,-20.881,444.766,174.706,17.738,152.821
C00669=1088.107,-21.132,444.779,174.704,17.737,152.821
C00670=1088.101,-21.381,444.792,174.703,17.735,152.821
C00671=1088.095,-21.631,444.805,174.701,17.733,152.821
C00672=1088.088,-21.880,444.818,174.699,17.731,152.821
C00673=1088.083,-22.129,444.830,174.698,17.730,152.821
C00674=1088.077,-22.379,444.843,174.696,17.729,152.821
C00675=1088.072,-22.629,444.857,174.695,17.727,152.821
C00676=1088.066,-22.879,444.869,174.693,17.725,152.821
C00677=1088.060,-23.128,444.883,174.691,17.723,152.821
C00678=1088.054,-23.378,444.895,174.690,17.722,152.821
C00679=1088.048,-23.628,444.908,174.688,17.720,152.821
C00680=1088.042,-23.876,444.921,174.687,17.719,152.821
C00681=1088.036,-24.126,444.933,174.686,17.717,152.821
C00682=1088.031,-24.376,444.946,174.683,17.715,152.821
C00683=1088.025,-24.625,444.960,174.682,17.714,152.821
C00684=1088.019,-24.875,444.972,174.680,17.712,152.821
C00685=1088.013,-25.125,444.985,174.679,17.711,152.821
C00686=1088.007,-25.374,444.998,174.678,17.709,152.821
C00687=1088.002,-25.624,445.010,174.675,17.707,152.821
C00688=1087.996,-25.874,445.023,174.674,17.705,152.821
C00689=1087.990,-26.123,445.035,174.673,17.704,152.821
C00690=1087.984,-26.373,445.049,174.671,17.703,152.821
C00691=1087.978,-26.623,445.062,174.670,17.701,152.821
C00692=1087.973,-26.872,445.074,174.668,17.700,152.821
C00693=1087.967,-27.121,445.087,174.666,17.697,152.821
C00694=1087.961,-27.371,445.100,174.665,17.696,152.821
C00695=1087.955,-27.621,445.112,174.663,17.694,152.821
C00696=1087.949,-27.871,445.125,174.662,17.693,152.821
C00697=1087.943,-28.120,445.138,174.660,17.692,152.821
C00698=1087.937,-28.370,445.151,174.659,17.690,152.821
C00699=1087.931,-28.619,445.162,174.657,17.688,152.821
C00700=1087.925,-28.869,445.175,174.655,17.686,152.821
C00701=1087.919,-29.119,445.187,174.654,17.685,152.821
C00702=1087.913,-29.368,445.201,174.652,17.684,152.821
C00703=1087.907,-29.618,445.213,174.651,17.682,152.821
C00704=1087.901,-29.868,445.226,174.649,17.681,152.821
C00705=1087.896,-30.117,445.238,174.648,17.679,152.821
C00706=1087.890,-30.367,445.250,174.646,17.677,152.821
C00707=1087.884,-30.616,445.264,174.644,17.676,152.821
C00708=1087.878,-30.866,445.276,174.643,17.674,152.821
C00709=1087.872,-31.116,445.289,174.641,17.673,152.821
C00710=1087.867,-31.365,445.301,174.640,17.671,152.821
C00711=1087.860,-31.615,445.313,174.638,17.670,152.821
C00712=1087.854,-31.865,445.325,174.636,17.668,152.821
C00713=1087.848,-32.114,445.338,174.635,17.666,152.821
C00714=1087.842,-32.363,445.351,174.633,17.665,152.821
C00715=1087.836,-32.635,445.364,174.632,17.663,152.821
C00716=1087.830,-32.906,445.378,174.630,17.661,152.821
C00717=1087.823,-33.177,445.392,174.628,17.660,152.821
C00718=1087.817,-33.448,445.406,174.627,17.658,152.821
C00719=1087.811,-33.697,445.418,174.625,17.657,152.821
C00720=1087.805,-33.947,445.430,174.624,17.655,152.821
C00721=1087.799,-34.197,445.443,174.622,17.653,152.821
C00722=1087.793,-34.447,445.455,174.620,17.651,152.821
C00723=1087.787,-34.696,445.467,174.619,17.650,152.821
C00724=1087.782,-34.946,445.480,174.617,17.649,152.821
C00725=1087.776,-35.196,445.492,174.616,17.647,152.821
C00726=1087.770,-35.445,445.504,174.615,17.646,152.821
C00727=1087.764,-35.695,445.517,174.613,17.644,152.821
C00728=1087.759,-35.945,445.529,174.611,17.642,152.821
C00729=1087.752,-36.194,445.541,174.609,17.641,152.821
C00730=1087.747,-36.443,445.554,174.608,17.639,152.821
C00731=1087.741,-36.693,445.566,174.607,17.638,152.821
C00732=1087.735,-36.943,445.579,174.605,17.636,152.821
C00733=1087.729,-37.192,445.591,174.604,17.635,152.821
C00734=1087.724,-37.442,445.603,174.602,17.633,152.821
C00735=1087.717,-37.692,445.615,174.601,17.632,152.821
C00736=1087.712,-37.941,445.628,174.599,17.630,152.821
C00737=1087.706,-38.191,445.640,174.597,17.628,152.821
C00738=1087.700,-38.441,445.653,174.596,17.627,152.821
C00739=1087.694,-38.690,445.665,174.594,17.625,152.821
C00740=1087.688,-38.940,445.677,174.593,17.624,152.821
C00741=1087.682,-39.189,445.689,174.591,17.622,152.820
C00742=1087.676,-39.439,445.702,174.590,17.621,152.821
C00743=1087.670,-39.689,445.713,174.588,17.620,152.821
C00744=1087.664,-39.939,445.725,174.586,17.618,152.821
C00745=1087.658,-40.189,445.738,174.585,17.616,152.821
C00746=1087.652,-40.437,445.749,174.583,17.615,152.821
C00747=1087.647,-40.687,445.762,174.582,17.613,152.821
C00748=1087.641,-40.937,445.775,174.580,17.612,152.821
C00749=1087.634,-41.187,445.787,174.579,17.611,152.821
C00750=1087.629,-41.436,445.799,174.577,17.609,152.821
C00751=1087.623,-41.686,445.811,174.576,17.607,152.821
C00752=1087.616,-41.936,445.823,174.574,17.606,152.821
C00753=1087.611,-42.185,445.835,174.572,17.604,152.821
C00754=1087.604,-42.435,445.847,174.571,17.603,152.821
C00755=1087.599,-42.685,445.859,174.569,17.601,152.821
C00756=1087.593,-42.934,445.871,174.568,17.600,152.821
C00757=1087.587,-43.184,445.883,174.566,17.598,152.821
C00758=1087.581,-43.434,445.895,174.565,17.597,152.821
C00759=1087.576,-43.683,445.907,174.563,17.596,152.821
C00760=1087.569,-43.933,445.919,174.562,17.594,152.821
C00761=1087.563,-44.183,445.932,174.561,17.593,152.821
C00762=1087.557,-44.432,445.943,174.558,17.591,152.821
C00763=1087.551,-44.682,445.955,174.557,17.589,152.821
C00764=1087.546,-44.931,445.968,174.555,17.588,152.821
C00765=1087.540,-45.181,445.979,174.554,17.586,152.821
C00766=1087.534,-45.431,445.992,174.552,17.585,152.821
C00767=1087.528,-45.680,446.003,174.551,17.584,152.821
C00768=1087.522,-45.930,446.015,174.550,17.582,152.821
C00769=1087.517,-46.179,446.028,174.548,17.581,152.821
C00770=1087.510,-46.429,446.039,174.547,17.579,152.821
C00771=1087.504,-46.679,446.051,174.545,17.578,152.821
C00772=1087.498,-46.928,446.063,174.543,17.577,152.821
C00773=1087.492,-47.178,446.076,174.541,17.575,152.821
C00774=1087.487,-47.427,446.086,174.540,17.573,152.821
C00775=1087.481,-47.677,446.099,174.538,17.572,152.821
C00776=1087.475,-47.927,446.112,174.537,17.570,152.821
C00777=1087.469,-48.177,446.122,174.535,17.569,152.821
C00778=1087.463,-48.427,446.135,174.534,17.567,152.821
C00779=1087.456,-48.698,446.148,174.532,17.566,152.821
C00780=1087.450,-48.969,446.161,174.531,17.564,152.821
C00781=1087.444,-49.240,446.174,174.529,17.562,152.821
C00782=1087.437,-49.512,446.186,174.527,17.561,152.821
C00783=1087.432,-49.762,446.198,174.526,17.560,152.821
C00784=1087.425,-50.011,446.210,174.524,17.558,152.821
C00785=1087.420,-50.262,446.222,174.523,17.556,152.821
C00786=1087.414,-50.511,446.233,174.521,17.555,152.821
C00787=1087.408,-50.761,446.245,174.520,17.554,152.821
C00788=1087.402,-51.010,446.257,174.518,17.553,152.821
C00789=1087.396,-51.260,446.269,174.516,17.551,152.821
C00790=1087.390,-51.510,446.281,174.515,17.550,152.821
C00791=1087.384,-51.759,446.292,174.513,17.548,152.821
C00792=1087.378,-52.009,446.304,174.512,17.546,152.821
C00793=1087.372,-52.258,446.316,174.510,17.545,152.821
C00794=1087.366,-52.508,446.328,174.509,17.544,152.821
C00795=1087.359,-52.758,446.339,174.507,17.543,152.821
C00796=1087.354,-53.007,446.351,174.506,17.541,152.821
C00797=1087.348,-53.257,446.362,174.504,17.540,152.821
C00798=1087.342,-53.506,446.374,174.503,17.538,152.821
C00799=1087.335,-53.756,446.385,174.501,17.537,152.821
C00800=1087.329,-54.006,446.398,174.500,17.536,152.821
C00801=1087.324,-54.256,446.409,174.498,17.534,152.821
C00802=1087.317,-54.505,446.421,174.497,17.533,152.821
C00803=1087.311,-54.755,446.431,174.495,17.531,152.821
C00804=1087.305,-55.005,446.444,174.494,17.530,152.821
C00805=1087.300,-55.254,446.455,174.492,17.529,152.821
C00806=1087.293,-55.504,446.467,174.491,17.528,152.821
C00807=1087.288,-55.754,446.478,174.489,17.526,152.821
C00808=1087.281,-56.003,446.490,174.487,17.525,152.822
C00809=1087.275,-56.253,446.502,174.485,17.523,152.822
C00810=1087.269,-56.502,446.513,174.484,17.522,152.822
C00811=1087.263,-56.753,446.525,174.482,17.520,152.822
C00812=1087.257,-57.002,446.537,174.481,17.519,152.822
C00813=1087.251,-57.252,446.548,174.479,17.518,152.822
C00814=1087.245,-57.501,446.559,174.478,17.517,152.822
C00815=1087.238,-57.751,446.571,174.476,17.515,152.822
C00816=1087.233,-58.001,446.582,174.475,17.513,152.822
C00817=1087.227,-58.250,446.594,174.473,17.512,152.822
C00818=1087.221,-58.500,446.605,174.472,17.511,152.822
C00819=1087.214,-58.749,446.617,174.470,17.510,152.822
C00820=1087.209,-58.999,446.628,174.469,17.508,152.822
C00821=1087.203,-59.249,446.640,174.467,17.507,152.822
C00822=1087.197,-59.498,446.651,174.466,17.505,152.822
C00823=1087.191,-59.748,446.662,174.464,17.504,152.822
C00824=1087.185,-59.998,446.673,174.463,17.503,152.822
C00825=1087.179,-60.248,446.686,174.461,17.502,152.822
C00826=1087.173,-60.497,446.697,174.460,17.500,152.822
C00827=1087.167,-60.747,446.708,174.458,17.499,152.822
C00828=1087.161,-60.996,446.720,174.457,17.497,152.822
C00829=1087.155,-61.246,446.730,174.455,17.496,152.822
C00830=1087.150,-61.496,446.742,174.454,17.495,152.822
C00831=1087.144,-61.745,446.754,174.452,17.494,152.822
C00832=1087.137,-61.995,446.765,174.451,17.492,152.822
C00833=1087.131,-62.245,446.776,174.449,17.491,152.822
C00834=1087.125,-62.494,446.788,174.448,17.489,152.822
C00835=1087.119,-62.744,446.799,174.446,17.488,152.822
C00836=1087.113,-62.994,446.811,174.445,17.487,152.822
C00837=1087.108,-63.244,446.822,174.443,17.486,152.822
C00838=1087.102,-63.493,446.833,174.442,17.484,152.822
C00839=1087.095,-63.743,446.844,174.440,17.483,152.823
C00840=1087.090,-63.992,446.855,174.439,17.481,152.822
C00841=1087.083,-64.243,446.867,174.437,17.480,152.823
C00842=1087.078,-64.492,446.879,174.436,17.479,152.823
C00843=1087.071,-64.765,446.890,174.433,17.477,152.823
C00844=1087.065,-65.037,446.903,174.432,17.476,152.823
C00845=1087.058,-65.310,446.916,174.430,17.474,152.823
C00846=1087.052,-65.583,446.927,174.429,17.473,152.823
C00847=1087.046,-65.833,446.938,174.427,17.472,152.823
C00848=1087.040,-66.082,446.951,174.426,17.470,152.823
C00849=1087.034,-66.332,446.961,174.424,17.469,152.823
C00850=1087.028,-66.582,446.973,174.423,17.468,152.823
C00851=1087.022,-66.832,446.984,174.421,17.466,152.823
C00852=1087.017,-67.081,446.994,174.419,17.465,152.823
C00853=1087.010,-67.331,447.006,174.418,17.464,152.823
C00854=1087.004,-67.580,447.017,174.416,17.463,152.823
C00855=1086.998,-67.830,447.028,174.415,17.461,152.823
C00856=1086.992,-68.080,447.039,174.413,17.460,152.823
C00857=1086.987,-68.330,447.051,174.412,17.458,152.823
C00858=1086.981,-68.580,447.062,174.410,17.457,152.823
C00859=1086.975,-68.829,447.073,174.409,17.456,152.823
C00860=1086.969,-69.079,447.084,174.407,17.455,152.823
C00861=1086.963,-69.329,447.095,174.406,17.453,152.823
C00862=1086.957,-69.578,447.107,174.404,17.452,152.823
C00863=1086.951,-69.827,447.118,174.403,17.451,152.824
C00864=1086.945,-70.077,447.128,174.401,17.449,152.824
C00865=1086.939,-70.327,447.140,174.399,17.448,152.824
C00866=1086.933,-70.576,447.151,174.398,17.447,152.824
C00867=1086.928,-70.826,447.161,174.396,17.446,152.824
C00868=1086.922,-71.076,447.173,174.395,17.444,152.824
C00869=1086.916,-71.326,447.184,174.393,17.443,152.824
C00870=1086.911,-71.575,447.195,174.392,17.442,152.824
C00871=1086.904,-71.826,447.206,174.390,17.440,152.824
C00872=1086.899,-72.075,447.217,174.389,17.439,152.824
C00873=1086.893,-72.325,447.228,174.387,17.438,152.824
C00874=1086.887,-72.574,447.239,174.386,17.437,152.824
C00875=1086.881,-72.824,447.250,174.384,17.435,152.824
C00876=1086.875,-73.074,447.261,174.383,17.434,152.824
C00877=1086.869,-73.323,447.272,174.381,17.433,152.824
C00878=1086.863,-73.573,447.283,174.380,17.431,152.824
C00879=1086.857,-73.823,447.294,174.378,17.430,152.824
C00880=1086.851,-74.072,447.305,174.377,17.429,152.824
C00881=1086.846,-74.322,447.316,174.375,17.428,152.824
C00882=1086.840,-74.571,447.327,174.373,17.426,152.824
C00883=1086.834,-74.822,447.338,174.373,17.425,152.824
C00884=1086.828,-75.071,447.349,174.371,17.424,152.824
C00885=1086.822,-75.321,447.360,174.370,17.423,152.825
C00886=1086.815,-75.570,447.370,174.368,17.422,152.825
C00887=1086.809,-75.820,447.381,174.366,17.421,152.825
C00888=1086.804,-76.069,447.392,174.365,17.420,152.825
C00889=1086.797,-76.320,447.403,174.363,17.418,152.825
C00890=1086.791,-76.569,447.414,174.362,17.417,152.825
C00891=1086.786,-76.819,447.425,174.360,17.416,152.825
C00892=1086.780,-77.068,447.436,174.359,17.415,152.825
C00893=1086.773,-77.319,447.446,174.357,17.413,152.825
C00894=1086.767,-77.568,447.457,174.355,17.412,152.825
C00895=1086.762,-77.818,447.468,174.354,17.411,152.825
C00896=1086.756,-78.067,447.478,174.352,17.410,152.825
C00897=1086.750,-78.317,447.490,174.351,17.408,152.825
C00898=1086.744,-78.567,447.501,174.349,17.407,152.825
C00899=1086.737,-78.816,447.511,174.348,17.406,152.826
C00900=1086.732,-79.065,447.522,174.346,17.405,152.826
C00901=1086.726,-79.316,447.532,174.345,17.404,152.826
C00902=1086.720,-79.566,447.543,174.344,17.403,152.826
C00903=1086.714,-79.815,447.554,174.342,17.402,152.826
C00904=1086.708,-80.064,447.564,174.341,17.400,152.826
C00905=1086.701,-80.315,447.576,174.339,17.399,152.826
C00906=1086.696,-80.564,447.586,174.337,17.398,152.826
C00907=1086.689,-80.839,447.598,174.336,17.397,152.826
C00908=1086.682,-81.114,447.609,174.334,17.396,152.826
C00909=1086.675,-81.389,447.621,174.332,17.395,152.826
C00910=1086.669,-81.664,447.633,174.330,17.393,152.826
C00911=1086.663,-81.914,447.644,174.329,17.392,152.826
C00912=1086.656,-82.164,447.654,174.328,17.391,152.826
C00913=1086.650,-82.413,447.665,174.326,17.390,152.827
C00914=1086.645,-82.663,447.675,174.324,17.389,152.827
C00915=1086.638,-82.913,447.686,174.323,17.388,152.827
C00916=1086.632,-83.163,447.697,174.321,17.386,152.827
C00917=1086.626,-83.412,447.708,174.320,17.385,152.827
C00918=1086.620,-83.662,447.717,174.318,17.384,152.827
C00919=1086.614,-83.911,447.728,174.316,17.383,152.827
C00920=1086.607,-84.161,447.739,174.315,17.382,152.827
C00921=1086.602,-84.411,447.750,174.313,17.381,152.827
C00922=1086.596,-84.661,447.760,174.312,17.380,152.827
C00923=1086.590,-84.910,447.770,174.311,17.379,152.827
C00924=1086.583,-85.160,447.781,174.309,17.378,152.827
C00925=1086.577,-85.410,447.791,174.308,17.377,152.828
C00926=1086.571,-85.659,447.802,174.306,17.376,152.828
C00927=1086.566,-85.909,447.813,174.304,17.375,152.828
C00928=1086.559,-86.158,447.823,174.303,17.373,152.828
C00929=1086.553,-86.409,447.833,174.301,17.372,152.828
C00930=1086.547,-86.658,447.844,174.299,17.371,152.828
C00931=1086.541,-86.908,447.855,174.298,17.370,152.828
C00932=1086.535,-87.158,447.865,174.297,17.369,152.828
C00933=1086.529,-87.407,447.875,174.296,17.368,152.828
C00934=1086.523,-87.658,447.886,174.294,17.367,152.828
C00935=1086.516,-87.907,447.896,174.292,17.366,152.828
C00936=1086.511,-88.156,447.907,174.291,17.365,152.829
C00937=1086.505,-88.406,447.917,174.289,17.364,152.829
C00938=1086.499,-88.656,447.927,174.287,17.363,152.829
C00939=1086.493,-88.905,447.938,174.286,17.362,152.829
C00940=1086.486,-89.156,447.948,174.285,17.361,152.829
C00941=1086.481,-89.405,447.959,174.283,17.360,152.829
C00942=1086.474,-89.655,447.968,174.282,17.359,152.829
C00943=1086.469,-89.904,447.979,174.280,17.357,152.829
C00944=1086.462,-90.154,447.990,174.279,17.356,152.829
C00945=1086.457,-90.404,448.000,174.277,17.355,152.829
C00946=1086.451,-90.653,448.011,174.275,17.354,152.830
C00947=1086.445,-90.903,448.020,174.274,17.353,152.830
C00948=1086.439,-91.153,448.031,174.273,17.353,152.830
C00949=1086.432,-91.403,448.041,174.271,17.351,152.830
C00950=1086.427,-91.652,448.052,174.269,17.350,152.830
C00951=1086.420,-91.902,448.061,174.268,17.349,152.830
C00952=1086.415,-92.152,448.072,174.266,17.348,152.830
C00953=1086.409,-92.402,448.082,174.264,17.347,152.830
C00954=1086.403,-92.651,448.093,174.263,17.346,152.830
C00955=1086.397,-92.901,448.102,174.261,17.345,152.830
C00956=1086.391,-93.150,448.113,174.260,17.344,152.831
C00957=1086.384,-93.401,448.123,174.259,17.343,152.831
C00958=1086.378,-93.650,448.134,174.257,17.342,152.831
C00959=1086.372,-93.900,448.144,174.255,17.341,152.831
C00960=1086.366,-94.150,448.154,174.254,17.340,152.831
C00961=1086.360,-94.399,448.164,174.252,17.339,152.831
C00962=1086.355,-94.649,448.175,174.250,17.338,152.831
C00963=1086.348,-94.899,448.184,174.250,17.337,152.831
C00964=1086.343,-95.148,448.195,174.248,17.336,152.831
C00965=1086.336,-95.398,448.205,174.246,17.335,152.831
C00966=1086.331,-95.647,448.216,174.245,17.334,152.832
C00967=1086.325,-95.897,448.225,174.243,17.333,152.832
C00968=1086.319,-96.147,448.236,174.242,17.332,152.832
C00969=1086.313,-96.397,448.246,174.241,17.331,152.832
C00970=1086.307,-96.647,448.256,174.239,17.330,152.832
C00971=1086.300,-96.924,448.267,174.237,17.329,152.832
C00972=1086.293,-97.201,448.279,174.236,17.328,152.832
C00973=1086.287,-97.478,448.290,174.234,17.327,152.832
C00974=1086.280,-97.755,448.301,174.232,17.326,152.832
C00975=1086.274,-98.005,448.311,174.231,17.325,152.833
C00976=1086.268,-98.255,448.322,174.229,17.324,152.833
C00977=1086.262,-98.504,448.331,174.227,17.323,152.833
C00978=1086.256,-98.754,448.341,174.226,17.322,152.833
C00979=1086.250,-99.004,448.352,174.224,17.321,152.833
C00980=1086.243,-99.254,448.362,174.223,17.320,152.833
C00981=1086.237,-99.504,448.371,174.222,17.319,152.833
C00982=1086.231,-99.754,448.382,174.220,17.319,152.833
C00983=1086.225,-100.003,448.392,174.218,17.318,152.834
C00984=1086.219,-100.253,448.401,174.216,17.316,152.834
C00985=1086.213,-100.502,448.411,174.215,17.315,152.834
C00986=1086.207,-100.752,448.422,174.214,17.315,152.834
C00987=1086.201,-101.002,448.431,174.212,17.314,152.834
C00988=1086.195,-101.251,448.441,174.211,17.313,152.834
C00989=1086.189,-101.502,448.452,174.209,17.312,152.834
C00990=1086.183,-101.751,448.461,174.207,17.311,152.834
C00991=1086.176,-102.001,448.472,174.206,17.311,152.835
C00992=1086.170,-102.250,448.481,174.205,17.309,152.835
C00993=1086.165,-102.500,448.491,174.203,17.308,152.835
C00994=1086.159,-102.750,448.501,174.201,17.307,152.835
C00995=1086.152,-102.999,448.511,174.200,17.306,152.835
C00996=1086.146,-103.249,448.521,174.199,17.306,152.835
C00997=1086.141,-103.499,448.531,174.197,17.305,152.835
C00998=1086.134,-103.749,448.540,174.195,17.304,152.835
C00999=1086.128,-103.998,448.551,174.194,17.303,152.836
C01000=1086.122,-104.248,448.560,174.192,17.302,152.836
C01001=1086.116,-104.498,448.570,174.191,17.302,152.836
C01002=1086.110,-104.748,448.580,174.189,17.301,152.836
C01003=1086.104,-104.998,448.590,174.188,17.300,152.836
C01004=1086.098,-105.247,448.600,174.186,17.299,152.836
C01005=1086.092,-105.497,448.610,174.184,17.298,152.836
C01006=1086.086,-105.747,448.620,174.183,17.298,152.837
C01007=1086.080,-105.997,448.629,174.181,17.297,152.837
C01008=1086.074,-106.246,448.639,174.180,17.295,152.837
C01009=1086.067,-106.496,448.649,174.178,17.294,152.837
C01010=1086.062,-106.746,448.659,174.177,17.293,152.837
C01011=1086.055,-106.996,448.669,174.175,17.293,152.837
C01012=1086.049,-107.245,448.678,174.174,17.292,152.837
C01013=1086.043,-107.495,448.688,174.172,17.291,152.837
C01014=1086.037,-107.745,448.697,174.170,17.290,152.838
C01015=1086.030,-107.994,448.708,174.169,17.290,152.838
C01016=1086.024,-108.244,448.717,174.168,17.289,152.838
C01017=1086.019,-108.494,448.727,174.166,17.288,152.838
C01018=1086.013,-108.744,448.737,174.164,17.287,152.838
C01019=1086.007,-108.994,448.747,174.163,17.286,152.838
C01020=1086.000,-109.243,448.756,174.162,17.286,152.838
C01021=1085.994,-109.493,448.766,174.160,17.285,152.839
C01022=1085.988,-109.743,448.775,174.158,17.284,152.839
C01023=1085.982,-109.993,448.785,174.156,17.283,152.839
C01024=1085.975,-110.242,448.795,174.155,17.283,152.839
C01025=1085.969,-110.492,448.805,174.154,17.282,152.839
C01026=1085.964,-110.741,448.814,174.152,17.281,152.839
C01027=1085.957,-110.991,448.823,174.150,17.280,152.840
C01028=1085.951,-111.240,448.833,174.149,17.280,152.840
C01029=1085.945,-111.490,448.843,174.148,17.279,152.840
C01030=1085.940,-111.740,448.853,174.146,17.278,152.840
C01031=1085.934,-111.990,448.862,174.144,17.277,152.840
C01032=1085.927,-112.240,448.872,174.143,17.276,152.840
C01033=1085.921,-112.490,448.881,174.141,17.276,152.841
C01034=1085.915,-112.740,448.891,174.140,17.275,152.841
C01035=1085.908,-113.012,448.902,174.138,17.274,152.841
C01036=1085.902,-113.284,448.911,174.136,17.273,152.841
C01037=1085.895,-113.557,448.922,174.134,17.272,152.841
C01038=1085.888,-113.830,448.932,174.133,17.272,152.841
C01039=1085.882,-114.079,448.942,174.132,17.271,152.841
C01040=1085.876,-114.328,448.951,174.130,17.270,152.842
C01041=1085.870,-114.578,448.961,174.128,17.269,152.842
C01042=1085.864,-114.828,448.970,174.126,17.268,152.842
C01043=1085.858,-115.078,448.980,174.125,17.268,152.842
C01044=1085.852,-115.328,448.989,174.124,17.267,152.842
C01045=1085.846,-115.577,448.999,174.122,17.266,152.842
C01046=1085.839,-115.827,449.009,174.121,17.266,152.843
C01047=1085.833,-116.077,449.018,174.119,17.265,152.843
C01048=1085.827,-116.327,449.028,174.117,17.265,152.843
C01049=1085.821,-116.577,449.037,174.116,17.263,152.843
C01050=1085.815,-116.826,449.047,174.115,17.263,152.843
C01051=1085.809,-117.075,449.056,174.113,17.262,152.843
C01052=1085.802,-117.325,449.065,174.111,17.262,152.844
C01053=1085.796,-117.575,449.075,174.109,17.261,152.844
C01054=1085.790,-117.825,449.084,174.109,17.260,152.844
C01055=1085.784,-118.074,449.094,174.107,17.260,152.844
C01056=1085.778,-118.324,449.103,174.105,17.259,152.844
C01057=1085.772,-118.575,449.112,174.104,17.259,152.844
C01058=1085.766,-118.824,449.122,174.102,17.258,152.845
C01059=1085.760,-119.073,449.131,174.100,17.257,152.845
C01060=1085.754,-119.323,449.141,174.099,17.256,152.845
C01061=1085.748,-119.573,449.150,174.098,17.256,152.845
C01062=1085.741,-119.823,449.159,174.096,17.255,152.845
C01063=1085.735,-120.072,449.169,174.094,17.254,152.846
C01064=1085.729,-120.323,449.177,174.093,17.254,152.846
C01065=1085.723,-120.573,449.187,174.091,17.253,152.846
C01066=1085.717,-120.822,449.196,174.089,17.253,152.846
C01067=1085.711,-121.071,449.206,174.088,17.252,152.846
C01068=1085.705,-121.321,449.215,174.087,17.252,152.846
C01069=1085.698,-121.571,449.225,174.085,17.250,152.847
C01070=1085.692,-121.821,449.233,174.083,17.250,152.847
C01071=1085.686,-122.071,449.243,174.082,17.249,152.847
C01072=1085.680,-122.320,449.252,174.080,17.249,152.847
C01073=1085.674,-122.570,449.262,174.079,17.248,152.847
C01074=1085.668,-122.820,449.271,174.078,17.248,152.848
C01075=1085.662,-123.070,449.280,174.076,17.247,152.848
C01076=1085.655,-123.320,449.289,174.074,17.246,152.848
C01077=1085.649,-123.569,449.298,174.072,17.246,152.848
C01078=1085.643,-123.818,449.308,174.071,17.245,152.848
C01079=1085.637,-124.068,449.317,174.069,17.244,152.849
C01080=1085.631,-124.319,449.326,174.068,17.243,152.849
C01081=1085.624,-124.568,449.335,174.067,17.243,152.849
C01082=1085.618,-124.818,449.345,174.065,17.243,152.849
C01083=1085.613,-125.067,449.354,174.063,17.242,152.849
C01084=1085.607,-125.317,449.363,174.062,17.242,152.849
C01085=1085.600,-125.567,449.372,174.060,17.241,152.850
C01086=1085.594,-125.817,449.381,174.058,17.240,152.850
C01087=1085.588,-126.067,449.390,174.057,17.240,152.850
C01088=1085.582,-126.316,449.399,174.056,17.239,152.850
C01089=1085.575,-126.566,449.408,174.054,17.238,152.850
C01090=1085.569,-126.816,449.418,174.053,17.238,152.851
C01091=1085.563,-127.066,449.427,174.051,17.237,152.851
C01092=1085.556,-127.315,449.436,174.049,17.237,152.851
C01093=1085.551,-127.565,449.445,174.048,17.237,152.851
C01094=1085.545,-127.815,449.454,174.046,17.236,152.851
C01095=1085.538,-128.072,449.464,174.044,17.235,152.852
C01096=1085.536,-128.329,449.474,174.043,17.234,152.852
C01097=1085.538,-128.585,449.486,174.042,17.230,152.851
C01098=1085.545,-128.838,449.499,174.042,17.227,152.850
C01099=1085.143,-128.859,449.369,173.999,17.340,152.880
C01100=1085.136,-128.606,449.355,174.000,17.344,152.881
C01101=1085.133,-128.351,449.343,174.000,17.348,152.881
C01102=1085.135,-128.094,449.332,174.001,17.350,152.882
C01103=1085.141,-127.837,449.323,174.002,17.350,152.881
C01104=1085.147,-127.587,449.314,174.004,17.350,152.881
C01105=1085.154,-127.338,449.305,174.006,17.351,152.881
C01106=1085.160,-127.088,449.296,174.007,17.351,152.881
C01107=1085.166,-126.838,449.286,174.009,17.352,152.880
C01108=1085.172,-126.589,449.277,174.011,17.353,152.880
C01109=1085.178,-126.339,449.269,174.012,17.353,152.880
C01110=1085.185,-126.089,449.259,174.013,17.354,152.880
C01111=1085.191,-125.839,449.250,174.015,17.355,152.880
C01112=1085.197,-125.589,449.242,174.016,17.355,152.880
C01113=1085.203,-125.339,449.232,174.018,17.356,152.879
C01114=1085.209,-125.090,449.223,174.020,17.356,152.879
C01115=1085.215,-124.840,449.213,174.021,17.356,152.879
C01116=1085.222,-124.590,449.205,174.023,17.357,152.879
C01117=1085.228,-124.340,449.195,174.025,17.358,152.879
C01118=1085.234,-124.090,449.186,174.025,17.358,152.878
C01119=1085.240,-123.841,449.177,174.027,17.359,152.878
C01120=1085.246,-123.591,449.168,174.029,17.360,152.878
C01121=1085.252,-123.341,449.159,174.031,17.361,152.878
C01122=1085.259,-123.092,449.149,174.032,17.361,152.878
C01123=1085.265,-122.842,449.140,174.034,17.362,152.878
C01124=1085.270,-122.593,449.130,174.036,17.362,152.877
C01125=1085.276,-122.342,449.122,174.037,17.363,152.877
C01126=1085.282,-122.093,449.112,174.038,17.363,152.877
C01127=1085.289,-121.843,449.103,174.040,17.364,152.877
C01128=1085.296,-121.593,449.093,174.041,17.364,152.877
C01129=1085.302,-121.343,449.084,174.043,17.365,152.876
C01130=1085.308,-121.093,449.075,174.045,17.366,152.876
C01131=1085.313,-120.844,449.066,174.046,17.367,152.876
C01132=1085.319,-120.594,449.056,174.048,17.367,152.876
C01133=1085.325,-120.344,449.047,174.049,17.368,152.876
C01134=1085.332,-120.095,449.038,174.051,17.369,152.875
C01135=1085.339,-119.845,449.028,174.052,17.369,152.875
C01136=1085.344,-119.595,449.019,174.054,17.370,152.875
C01137=1085.350,-119.346,449.010,174.056,17.371,152.875
C01138=1085.356,-119.096,449.001,174.057,17.372,152.875
C01139=1085.362,-118.846,448.991,174.058,17.372,152.875
C01140=1085.369,-118.596,448.981,174.060,17.373,152.875
C01141=1085.375,-118.346,448.972,174.062,17.373,152.874
C01142=1085.381,-118.097,448.962,174.064,17.375,152.874
C01143=1085.388,-117.847,448.953,174.065,17.375,152.874
C01144=1085.394,-117.597,448.944,174.066,17.376,152.874
C01145=1085.400,-117.348,448.935,174.068,17.376,152.874
C01146=1085.405,-117.098,448.926,174.069,17.377,152.874
C01147=1085.412,-116.848,448.916,174.071,17.378,152.873
C01148=1085.418,-116.598,448.907,174.073,17.378,152.873
C01149=1085.424,-116.348,448.897,174.074,17.379,152.873
C01150=1085.430,-116.099,448.887,174.075,17.379,152.873
C01151=1085.436,-115.849,448.878,174.077,17.380,152.873
C01152=1085.442,-115.599,448.868,174.079,17.381,152.872
C01153=1085.449,-115.349,448.859,174.081,17.382,152.872
C01154=1085.455,-115.099,448.849,174.081,17.383,152.872
C01155=1085.460,-114.850,448.840,174.083,17.383,152.872
C01156=1085.466,-114.600,448.830,174.085,17.384,152.872
C01157=1085.473,-114.351,448.821,174.087,17.385,152.872
C01158=1085.479,-114.101,448.811,174.088,17.385,152.872
C01159=1085.485,-113.851,448.802,174.089,17.386,152.871
C01160=1085.492,-113.578,448.792,174.091,17.387,152.871
C01161=1085.498,-113.306,448.781,174.093,17.388,152.871
C01162=1085.505,-113.033,448.771,174.095,17.389,152.871
C01163=1085.512,-112.760,448.760,174.097,17.390,152.871
C01164=1085.519,-112.511,448.750,174.098,17.391,152.871
C01165=1085.524,-112.261,448.740,174.099,17.391,152.871
C01166=1085.530,-112.011,448.731,174.101,17.392,152.870
C01167=1085.536,-111.762,448.721,174.103,17.393,152.870
C01168=1085.542,-111.512,448.712,174.104,17.394,152.870
C01169=1085.548,-111.262,448.702,174.105,17.394,152.870
C01170=1085.554,-111.012,448.693,174.107,17.395,152.870
C01171=1085.560,-110.762,448.683,174.109,17.396,152.870
C01172=1085.567,-110.513,448.674,174.110,17.397,152.869
C01173=1085.573,-110.263,448.664,174.111,17.397,152.869
C01174=1085.579,-110.013,448.654,174.113,17.398,152.869
C01175=1085.585,-109.763,448.645,174.115,17.399,152.869
C01176=1085.591,-109.513,448.635,174.117,17.400,152.869
C01177=1085.597,-109.264,448.626,174.117,17.400,152.869
C01178=1085.604,-109.014,448.615,174.119,17.401,152.869
C01179=1085.609,-108.764,448.605,174.121,17.403,152.868
C01180=1085.616,-108.515,448.596,174.123,17.403,152.868
C01181=1085.622,-108.265,448.586,174.124,17.404,152.868
C01182=1085.628,-108.015,448.577,174.125,17.405,152.868
C01183=1085.634,-107.765,448.567,174.127,17.406,152.868
C01184=1085.640,-107.515,448.557,174.129,17.406,152.868
C01185=1085.647,-107.266,448.547,174.130,17.407,152.868
C01186=1085.653,-107.016,448.538,174.131,17.408,152.867
C01187=1085.658,-106.766,448.527,174.133,17.409,152.867
C01188=1085.664,-106.517,448.518,174.135,17.410,152.867
C01189=1085.671,-106.267,448.508,174.136,17.411,152.867
C01190=1085.677,-106.017,448.499,174.138,17.412,152.867
C01191=1085.683,-105.768,448.488,174.139,17.412,152.867
C01192=1085.689,-105.518,448.478,174.141,17.413,152.867
C01193=1085.694,-105.269,448.469,174.142,17.414,152.867
C01194=1085.700,-105.019,448.460,174.144,17.415,152.866
C01195=1085.707,-104.769,448.450,174.146,17.416,152.866
C01196=1085.712,-104.519,448.439,174.147,17.416,152.866
C01197=1085.719,-104.270,448.430,174.148,17.418,152.866
C01198=1085.725,-104.020,448.420,174.150,17.419,152.866
C01199=1085.731,-103.770,448.410,174.152,17.420,152.866
C01200=1085.737,-103.521,448.400,174.153,17.421,152.866
C01201=1085.743,-103.271,448.390,174.154,17.421,152.865
C01202=1085.749,-103.021,448.380,174.156,17.422,152.865
C01203=1085.755,-102.771,448.371,174.158,17.423,152.865
C01204=1085.761,-102.521,448.360,174.159,17.424,152.865
C01205=1085.768,-102.271,448.350,174.161,17.425,152.865
C01206=1085.774,-102.021,448.340,174.163,17.426,152.865
C01207=1085.780,-101.772,448.331,174.163,17.427,152.865
C01208=1085.786,-101.522,448.320,174.165,17.428,152.865
C01209=1085.792,-101.272,448.310,174.167,17.429,152.865
C01210=1085.798,-101.022,448.301,174.169,17.429,152.864
C01211=1085.805,-100.773,448.291,174.170,17.430,152.864
C01212=1085.810,-100.523,448.280,174.171,17.431,152.864
C01213=1085.816,-100.273,448.271,174.173,17.432,152.864
C01214=1085.823,-100.024,448.261,174.174,17.433,152.864
C01215=1085.828,-99.774,448.250,174.176,17.434,152.864
C01216=1085.834,-99.524,448.241,174.178,17.435,152.864
C01217=1085.841,-99.275,448.231,174.179,17.436,152.864
C01218=1085.847,-99.025,448.221,174.180,17.437,152.864
C01219=1085.852,-98.775,448.211,174.182,17.438,152.863
C01220=1085.859,-98.526,448.201,174.184,17.439,152.863
C01221=1085.865,-98.276,448.191,174.186,17.439,152.863
C01222=1085.871,-98.027,448.180,174.187,17.441,152.863
C01223=1085.877,-97.776,448.170,174.189,17.442,152.863
C01224=1085.884,-97.499,448.159,174.190,17.443,152.863
C01225=1085.891,-97.221,448.148,174.192,17.444,152.863
C01226=1085.897,-96.945,448.137,174.194,17.445,152.862
C01227=1085.904,-96.667,448.125,174.195,17.446,152.862
C01228=1085.910,-96.417,448.115,174.197,17.447,152.862
C01229=1085.915,-96.167,448.105,174.198,17.447,152.862
C01230=1085.922,-95.917,448.095,174.199,17.449,152.862
C01231=1085.928,-95.668,448.085,174.201,17.450,152.862
C01232=1085.934,-95.418,448.075,174.203,17.451,152.862
C01233=1085.940,-95.169,448.064,174.204,17.452,152.862
C01234=1085.945,-94.919,448.054,174.206,17.453,152.862
C01235=1085.952,-94.670,448.044,174.208,17.454,152.862
C01236=1085.957,-94.420,448.034,174.208,17.455,152.862
C01237=1085.964,-94.170,448.024,174.210,17.456,152.862
C01238=1085.969,-93.920,448.013,174.212,17.457,152.861
C01239=1085.975,-93.671,448.004,174.213,17.458,152.861
C01240=1085.982,-93.420,447.992,174.215,17.459,152.861
C01241=1085.987,-93.170,447.982,174.217,17.460,152.861
C01242=1085.994,-92.921,447.972,174.218,17.461,152.861
C01243=1085.999,-92.671,447.962,174.220,17.462,152.861
C01244=1086.006,-92.422,447.951,174.221,17.463,152.861
C01245=1086.011,-92.172,447.941,174.222,17.465,152.861
C01246=1086.018,-91.922,447.931,174.224,17.466,152.861
C01247=1086.023,-91.673,447.920,174.225,17.467,152.861
C01248=1086.029,-91.423,447.911,174.227,17.468,152.860
C01249=1086.035,-91.174,447.900,174.229,17.469,152.860
C01250=1086.042,-90.923,447.890,174.230,17.470,152.860
C01251=1086.048,-90.674,447.879,174.231,17.470,152.860
C01252=1086.054,-90.424,447.869,174.233,17.472,152.860
C01253=1086.060,-90.174,447.858,174.235,17.473,152.860
C01254=1086.066,-89.925,447.849,174.236,17.474,152.860
C01255=1086.071,-89.675,447.838,174.238,17.475,152.860
C01256=1086.077,-89.426,447.827,174.239,17.476,152.860
C01257=1086.084,-89.175,447.817,174.241,17.477,152.860
C01258=1086.090,-88.926,447.806,174.243,17.478,152.860
C01259=1086.096,-88.676,447.797,174.244,17.480,152.859
C01260=1086.102,-88.426,447.786,174.245,17.480,152.859
C01261=1086.108,-88.177,447.776,174.247,17.481,152.859
C01262=1086.114,-87.927,447.765,174.248,17.483,152.859
C01263=1086.119,-87.678,447.755,174.250,17.484,152.859
C01264=1086.126,-87.428,447.744,174.251,17.485,152.859
C01265=1086.132,-87.178,447.734,174.253,17.486,152.859
C01266=1086.138,-86.928,447.723,174.255,17.487,152.859
C01267=1086.144,-86.679,447.713,174.256,17.488,152.859
C01268=1086.149,-86.429,447.702,174.258,17.489,152.859
C01269=1086.157,-86.179,447.692,174.259,17.490,152.859
C01270=1086.162,-85.929,447.681,174.260,17.491,152.859
C01271=1086.168,-85.680,447.671,174.262,17.492,152.858
C01272=1086.174,-85.430,447.660,174.263,17.493,152.858
C01273=1086.180,-85.181,447.650,174.265,17.494,152.858
C01274=1086.187,-84.930,447.640,174.267,17.496,152.858
C01275=1086.192,-84.681,447.629,174.268,17.497,152.858
C01276=1086.199,-84.432,447.619,174.270,17.498,152.858
C01277=1086.205,-84.182,447.608,174.271,17.499,152.858
C01278=1086.211,-83.931,447.597,174.273,17.500,152.858
C01279=1086.217,-83.682,447.587,174.275,17.501,152.858
C01280=1086.223,-83.433,447.576,174.275,17.502,152.858
C01281=1086.229,-83.183,447.566,174.277,17.504,152.858
C01282=1086.235,-82.933,447.555,174.279,17.505,152.858
C01283=1086.241,-82.683,447.544,174.280,17.506,152.858
C01284=1086.248,-82.434,447.534,174.282,17.507,152.857
C01285=1086.253,-82.184,447.523,174.283,17.508,152.857
C01286=1086.259,-81.934,447.513,174.285,17.509,152.857
C01287=1086.266,-81.684,447.502,174.287,17.510,152.857
C01288=1086.272,-81.409,447.490,174.288,17.512,152.857
C01289=1086.279,-81.135,447.479,174.290,17.513,152.857
C01290=1086.286,-80.860,447.467,174.291,17.514,152.857
C01291=1086.292,-80.584,447.455,174.293,17.515,152.857
C01292=1086.299,-80.334,447.445,174.295,17.516,152.857
C01293=1086.305,-80.085,447.434,174.296,17.517,152.857
C01294=1086.311,-79.835,447.423,174.298,17.519,152.857
C01295=1086.317,-79.585,447.412,174.299,17.520,152.857
C01296=1086.323,-79.335,447.401,174.301,17.521,152.856
C01297=1086.329,-79.086,447.391,174.302,17.523,152.857
C01298=1086.335,-78.836,447.381,174.304,17.524,152.856
C01299=1086.341,-78.586,447.369,174.306,17.525,152.856
C01300=1086.347,-78.336,447.358,174.307,17.526,152.856
C01301=1086.352,-78.087,447.348,174.309,17.527,152.856
C01302=1086.359,-77.838,447.337,174.310,17.529,152.856
C01303=1086.365,-77.588,447.326,174.312,17.530,152.856
C01304=1086.371,-77.338,447.315,174.313,17.531,152.856
C01305=1086.377,-77.089,447.304,174.314,17.532,152.856
C01306=1086.382,-76.839,447.294,174.316,17.533,152.856
C01307=1086.388,-76.588,447.283,174.317,17.534,152.856
C01308=1086.394,-76.339,447.272,174.319,17.535,152.856
C01309=1086.401,-76.090,447.262,174.320,17.537,152.856
C01310=1086.407,-75.839,447.250,174.322,17.538,152.856
C01311=1086.413,-75.590,447.240,174.324,17.539,152.856
C01312=1086.418,-75.340,447.229,174.325,17.541,152.856
C01313=1086.424,-75.091,447.218,174.327,17.542,152.856
C01314=1086.431,-74.841,447.207,174.328,17.543,152.855
C01315=1086.436,-74.591,447.196,174.330,17.544,152.855
C01316=1086.443,-74.342,447.185,174.331,17.546,152.855
C01317=1086.449,-74.092,447.174,174.333,17.547,152.855
C01318=1086.455,-73.842,447.163,174.334,17.548,152.855
C01319=1086.461,-73.593,447.152,174.336,17.549,152.855
C01320=1086.466,-73.343,447.142,174.337,17.551,152.855
C01321=1086.472,-73.093,447.130,174.339,17.552,152.855
C01322=1086.478,-72.843,447.119,174.340,17.554,152.855
C01323=1086.483,-72.594,447.108,174.342,17.555,152.855
C01324=1086.489,-72.345,447.097,174.343,17.556,152.855
C01325=1086.495,-72.094,447.086,174.345,17.557,152.855
C01326=1086.501,-71.845,447.075,174.346,17.559,152.855
C01327=1086.507,-71.595,447.064,174.348,17.560,152.855
C01328=1086.513,-71.345,447.053,174.350,17.561,152.855
C01329=1086.519,-71.096,447.042,174.351,17.563,152.855
C01330=1086.525,-70.846,447.031,174.353,17.564,152.855
C01331=1086.530,-70.597,447.020,174.354,17.565,152.855
C01332=1086.537,-70.346,447.009,174.356,17.566,152.855
C01333=1086.543,-70.097,446.998,174.357,17.568,152.855
C01334=1086.549,-69.848,446.986,174.359,17.569,152.855
C01335=1086.555,-69.598,446.975,174.360,17.571,152.855
C01336=1086.560,-69.348,446.964,174.362,17.572,152.855
C01337=1086.566,-69.099,446.953,174.363,17.573,152.855
C01338=1086.572,-68.848,446.942,174.365,17.574,152.854
C01339=1086.578,-68.599,446.931,174.366,17.576,152.854
C01340=1086.584,-68.349,446.920,174.368,17.577,152.854
C01341=1086.590,-68.099,446.909,174.369,17.578,152.854
C01342=1086.596,-67.850,446.898,174.371,17.580,152.854
C01343=1086.602,-67.601,446.886,174.372,17.581,152.854
C01344=1086.608,-67.351,446.875,174.374,17.582,152.854
C01345=1086.613,-67.101,446.863,174.375,17.584,152.854
C01346=1086.619,-66.851,446.853,174.377,17.585,152.854
C01347=1086.625,-66.601,446.841,174.378,17.586,152.854
C01348=1086.631,-66.352,446.830,174.380,17.588,152.854
C01349=1086.637,-66.102,446.818,174.381,17.589,152.854
C01350=1086.643,-65.853,446.808,174.383,17.591,152.854
C01351=1086.649,-65.603,446.797,174.385,17.592,152.854
C01352=1086.656,-65.330,446.784,174.386,17.593,152.854
C01353=1086.662,-65.057,446.772,174.388,17.594,152.854
C01354=1086.669,-64.785,446.760,174.389,17.596,152.854
C01355=1086.675,-64.511,446.747,174.391,17.597,152.854
C01356=1086.681,-64.262,446.737,174.392,17.599,152.854
C01357=1086.687,-64.012,446.725,174.394,17.600,152.854
C01358=1086.692,-63.762,446.713,174.395,17.601,152.854
C01359=1086.699,-63.512,446.702,174.396,17.603,152.854
C01360=1086.704,-63.263,446.691,174.398,17.604,152.854
C01361=1086.710,-63.014,446.679,174.399,17.606,152.854
C01362=1086.717,-62.763,446.668,174.401,17.607,152.854
C01363=1086.722,-62.514,446.657,174.402,17.608,152.854
C01364=1086.728,-62.264,446.645,174.404,17.609,152.854
C01365=1086.734,-62.015,446.634,174.406,17.611,152.854
C01366=1086.740,-61.764,446.623,174.408,17.612,152.854
C01367=1086.747,-61.516,446.611,174.409,17.614,152.854
C01368=1086.753,-61.265,446.600,174.411,17.615,152.854
C01369=1086.758,-61.016,446.588,174.412,17.617,152.854
C01370=1086.764,-60.767,446.577,174.414,17.618,152.854
C01371=1086.770,-60.516,446.565,174.415,17.619,152.853
C01372=1086.776,-60.267,446.555,174.417,17.621,152.854
C01373=1086.783,-60.017,446.543,174.418,17.622,152.853
C01374=1086.788,-59.768,446.531,174.420,17.624,152.853
C01375=1086.794,-59.517,446.520,174.422,17.625,152.853
C01376=1086.800,-59.269,446.508,174.423,17.626,152.853
C01377=1086.806,-59.018,446.497,174.424,17.628,152.853
C01378=1086.812,-58.769,446.486,174.426,17.629,152.853
C01379=1086.818,-58.519,446.474,174.427,17.630,152.853
C01380=1086.824,-58.269,446.463,174.429,17.632,152.853
C01381=1086.830,-58.020,446.451,174.430,17.633,152.853
C01382=1086.836,-57.770,446.440,174.432,17.634,152.853
C01383=1086.842,-57.521,446.427,174.433,17.636,152.853
C01384=1086.848,-57.271,446.416,174.435,17.637,152.853
C01385=1086.854,-57.021,446.405,174.436,17.638,152.853
C01386=1086.860,-56.772,446.394,174.438,17.640,152.853
C01387=1086.866,-56.521,446.382,174.439,17.641,152.853
C01388=1086.872,-56.273,446.370,174.441,17.643,152.853
C01389=1086.878,-56.022,446.359,174.442,17.644,152.853
C01390=1086.885,-55.773,446.347,174.444,17.645,152.853
C01391=1086.890,-55.523,446.336,174.445,17.647,152.853
C01392=1086.896,-55.273,446.324,174.447,17.648,152.853
C01393=1086.902,-55.024,446.313,174.449,17.650,152.853
C01394=1086.909,-54.774,446.301,174.451,17.651,152.853
C01395=1086.914,-54.525,446.289,174.452,17.653,152.853
C01396=1086.920,-54.275,446.277,174.454,17.654,152.853
C01397=1086.927,-54.025,446.266,174.455,17.655,152.853
C01398=1086.933,-53.776,446.254,174.457,17.657,152.853
C01399=1086.938,-53.525,446.243,174.458,17.658,152.853
C01400=1086.945,-53.277,446.231,174.460,17.660,152.853
C01401=1086.951,-53.026,446.220,174.461,17.661,152.853
C01402=1086.956,-52.777,446.208,174.463,17.662,152.853
C01403=1086.963,-52.528,446.196,174.464,17.664,152.853
C01404=1086.969,-52.277,446.184,174.465,17.665,152.853
C01405=1086.975,-52.029,446.173,174.467,17.666,152.853
C01406=1086.981,-51.778,446.161,174.469,17.668,152.853
C01407=1086.987,-51.529,446.149,174.470,17.669,152.853
C01408=1086.993,-51.279,446.138,174.472,17.671,152.853
C01409=1086.999,-51.029,446.126,174.473,17.672,152.853
C01410=1087.005,-50.780,446.114,174.475,17.674,152.853
C01411=1087.011,-50.530,446.103,174.477,17.675,152.853
C01412=1087.017,-50.280,446.090,174.478,17.677,152.853
C01413=1087.023,-50.031,446.079,174.480,17.678,152.853
C01414=1087.029,-49.781,446.067,174.481,17.680,152.853
C01415=1087.035,-49.532,446.055,174.483,17.681,152.853
C01416=1087.041,-49.260,446.042,174.484,17.683,152.853
C01417=1087.047,-48.988,446.029,174.486,17.684,152.853
C01418=1087.054,-48.716,446.016,174.488,17.686,152.853
C01419=1087.061,-48.445,446.003,174.489,17.688,152.853
C01420=1087.066,-48.195,445.992,174.491,17.689,152.853
C01421=1087.072,-47.945,445.979,174.492,17.690,152.853
C01422=1087.078,-47.696,445.967,174.494,17.692,152.853
C01423=1087.084,-47.447,445.955,174.495,17.693,152.853
C01424=1087.090,-47.196,445.944,174.496,17.695,152.853
C01425=1087.095,-46.947,445.932,174.499,17.697,152.853
C01426=1087.102,-46.698,445.920,174.500,17.698,152.853
C01427=1087.107,-46.448,445.908,174.502,17.700,152.853
C01428=1087.113,-46.198,445.896,174.503,17.701,152.853
C01429=1087.120,-45.948,445.884,174.505,17.702,152.853
C01430=1087.125,-45.699,445.872,174.506,17.704,152.853
C01431=1087.131,-45.449,445.860,174.508,17.706,152.853
C01432=1087.137,-45.199,445.848,174.509,17.707,152.853
C01433=1087.143,-44.950,445.836,174.510,17.709,152.853
C01434=1087.149,-44.700,445.824,174.512,17.710,152.853
C01435=1087.154,-44.451,445.812,174.513,17.711,152.853
C01436=1087.161,-44.201,445.800,174.516,17.714,152.853
C01437=1087.167,-43.951,445.788,174.517,17.715,152.853
C01438=1087.173,-43.702,445.776,174.519,17.716,152.853
C01439=1087.179,-43.452,445.763,174.520,17.718,152.853
C01440=1087.184,-43.202,445.752,174.521,17.719,152.853
C01441=1087.190,-42.953,445.740,174.523,17.721,152.853
C01442=1087.196,-42.703,445.728,174.524,17.722,152.853
C01443=1087.202,-42.453,445.715,174.526,17.724,152.853
C01444=1087.208,-42.204,445.703,174.527,17.725,152.853
C01445=1087.214,-41.955,445.691,174.529,17.727,152.853
C01446=1087.220,-41.704,445.679,174.531,17.728,152.853
C01447=1087.226,-41.455,445.667,174.532,17.730,152.853
C01448=1087.232,-41.205,445.655,174.534,17.731,152.853
C01449=1087.238,-40.956,445.643,174.535,17.733,152.853
C01450=1087.243,-40.707,445.631,174.537,17.735,152.853
C01451=1087.249,-40.457,445.618,174.538,17.736,152.853
C01452=1087.256,-40.207,445.606,174.540,17.737,152.853
C01453=1087.262,-39.957,445.594,174.541,17.739,152.853
C01454=1087.267,-39.707,445.582,174.543,17.741,152.853
C01455=1087.274,-39.458,445.570,174.545,17.742,152.853
C01456=1087.279,-39.208,445.558,174.546,17.744,152.853
C01457=1087.285,-38.959,445.545,174.548,17.745,152.853
C01458=1087.291,-38.709,445.533,174.549,17.747,152.853
C01459=1087.297,-38.459,445.521,174.550,17.748,152.853
C01460=1087.303,-38.209,445.508,174.552,17.749,152.853
C01461=1087.309,-37.960,445.496,174.553,17.751,152.853
C01462=1087.314,-37.710,445.484,174.556,17.753,152.853
C01463=1087.321,-37.461,445.472,174.557,17.755,152.853
C01464=1087.326,-37.212,445.459,174.558,17.756,152.853
C01465=1087.332,-36.962,445.447,174.560,17.758,152.853
C01466=1087.338,-36.712,445.434,174.561,17.759,152.853
C01467=1087.344,-36.463,445.422,174.563,17.760,152.853
C01468=1087.349,-36.213,445.410,174.564,17.762,152.853
C01469=1087.355,-35.963,445.397,174.566,17.764,152.853
C01470=1087.361,-35.714,445.385,174.568,17.766,152.853
C01471=1087.367,-35.464,445.373,174.569,17.767,152.853
C01472=1087.373,-35.214,445.360,174.571,17.769,152.853
C01473=1087.379,-34.964,445.348,174.572,17.771,152.853
C01474=1087.384,-34.715,445.336,174.574,17.772,152.853
C01475=1087.390,-34.465,445.323,174.575,17.773,152.853
C01476=1087.396,-34.215,445.311,174.577,17.775,152.853
C01477=1087.403,-33.966,445.299,174.579,17.777,152.853
C01478=1087.408,-33.717,445.286,174.580,17.778,152.853
C01479=1087.414,-33.467,445.274,174.581,17.780,152.853
C01480=1087.421,-33.196,445.260,174.583,17.782,152.853
C01481=1087.427,-32.924,445.247,174.585,17.784,152.853
C01482=1087.434,-32.653,445.233,174.586,17.785,152.853
C01483=1087.440,-32.381,445.219,174.588,17.787,152.853
C01484=1087.445,-32.132,445.207,174.589,17.788,152.853
C01485=1087.451,-31.882,445.195,174.592,17.790,152.853
C01486=1087.457,-31.633,445.181,174.593,17.792,152.853
C01487=1087.463,-31.383,445.169,174.594,17.793,152.853
C01488=1087.469,-31.133,445.156,174.596,17.795,152.853
C01489=1087.475,-30.884,445.144,174.597,17.796,152.853
C01490=1087.481,-30.635,445.132,174.599,17.798,152.853
C01491=1087.487,-30.385,445.119,174.601,17.800,152.853
C01492=1087.493,-30.135,445.107,174.603,17.801,152.853
C01493=1087.499,-29.886,445.094,174.604,17.803,152.853
C01494=1087.505,-29.636,445.081,174.605,17.804,152.853
C01495=1087.510,-29.387,445.069,174.607,17.806,152.853
C01496=1087.516,-29.137,445.056,174.608,17.807,152.853
C01497=1087.522,-28.887,445.044,174.609,17.809,152.853
C01498=1087.528,-28.637,445.030,174.612,17.811,152.853
C01499=1087.534,-28.388,445.018,174.613,17.812,152.853
C01500=1087.540,-28.138,445.006,174.615,17.814,152.853
C01501=1087.546,-27.889,444.993,174.616,17.815,152.853
C01502=1087.552,-27.639,444.980,174.618,17.817,152.853
C01503=1087.558,-27.389,444.967,174.619,17.818,152.853
C01504=1087.564,-27.140,444.955,174.621,17.821,152.853
C01505=1087.570,-26.890,444.942,174.623,17.822,152.854
C01506=1087.576,-26.640,444.929,174.624,17.823,152.853
C01507=1087.581,-26.391,444.917,174.626,17.825,152.853
C01508=1087.587,-26.141,444.904,174.627,17.826,152.853
C01509=1087.593,-25.892,444.891,174.629,17.828,152.853
C01510=1087.599,-25.642,444.878,174.631,17.830,152.854
C01511=1087.605,-25.392,444.866,174.632,17.832,152.854
C01512=1087.611,-25.144,444.853,174.633,17.833,152.854
C01513=1087.617,-24.894,444.840,174.635,17.835,152.854
C01514=1087.622,-24.644,444.827,174.636,17.836,152.854
C01515=1087.628,-24.394,444.814,174.638,17.838,152.854
C01516=1087.634,-24.144,444.801,174.640,17.840,152.854
C01517=1087.640,-23.895,444.789,174.641,17.842,152.854
C01518=1087.646,-23.645,444.776,174.642,17.843,152.854
C01519=1087.651,-23.396,444.763,174.644,17.845,152.854
C01520=1087.657,-23.146,444.751,174.646,17.847,152.854
C01521=1087.663,-22.897,444.737,174.647,17.848,152.854
C01522=1087.669,-22.647,444.724,174.649,17.850,152.854
C01523=1087.674,-22.397,444.712,174.651,17.851,152.854
C01524=1087.681,-22.148,444.699,174.652,17.853,152.854
C01525=1087.687,-21.898,444.686,174.653,17.854,152.854
C01526=1087.693,-21.649,444.673,174.656,17.856,152.854
C01527=1087.697,-21.399,444.660,174.657,17.858,152.854
C01528=1087.704,-21.150,444.647,174.658,17.860,152.854
C01529=1087.709,-20.900,444.634,174.660,17.861,152.854
C01530=1087.715,-20.650,444.622,174.661,17.863,152.854
C01531=1087.722,-20.401,444.608,174.663,17.865,152.854
C01532=1087.728,-20.151,444.596,174.665,17.866,152.854
C01533=1087.733,-19.901,444.582,174.666,17.868,152.854
C01534=1087.739,-19.651,444.569,174.667,17.870,152.854
C01535=1087.745,-19.402,444.556,174.669,17.871,152.854
C01536=1087.751,-19.152,444.544,174.671,17.873,152.854
C01537=1087.757,-18.903,444.530,174.672,17.875,152.854
C01538=1087.762,-18.653,444.517,174.674,17.876,152.854
C01539=1087.769,-18.404,444.504,174.676,17.877,152.854
C01540=1087.775,-18.154,444.491,174.677,17.879,152.854
C01541=1087.780,-17.905,444.478,174.679,17.881,152.854
C01542=1087.785,-17.655,444.465,174.681,17.883,152.854
C01543=1087.792,-17.406,444.452,174.682,17.884,152.854
C01544=1087.798,-17.133,444.438,174.683,17.886,152.854
C01545=1087.805,-16.861,444.423,174.686,17.888,152.854
C01546=1087.811,-16.589,444.409,174.687,17.890,152.855
C01547=1087.818,-16.318,444.395,174.689,17.892,152.855
C01548=1087.823,-16.067,444.382,174.691,17.893,152.855
C01549=1087.829,-15.818,444.369,174.692,17.895,152.855
C01550=1087.835,-15.568,444.356,174.693,17.896,152.855
C01551=1087.841,-15.319,444.343,174.695,17.898,152.855
C01552=1087.847,-15.069,444.329,174.697,17.900,152.855
C01553=1087.853,-14.819,444.316,174.698,17.902,152.855
C01554=1087.859,-14.570,444.303,174.700,17.903,152.855
C01555=1087.864,-14.321,444.289,174.701,17.905,152.855
C01556=1087.870,-14.071,444.277,174.703,17.907,152.855
C01557=1087.876,-13.821,444.263,174.705,17.908,152.855
C01558=1087.882,-13.571,444.250,174.706,17.910,152.855
C01559=1087.888,-13.322,444.237,174.708,17.912,152.855
C01560=1087.893,-13.072,444.223,174.709,17.913,152.855
C01561=1087.899,-12.823,444.211,174.711,17.915,152.855
C01562=1087.905,-12.573,444.197,174.713,17.917,152.855
C01563=1087.911,-12.324,444.184,174.714,17.918,152.855
C01564=1087.917,-12.074,444.170,174.715,17.920,152.855
C01565=1087.922,-11.824,444.157,174.718,17.922,152.855
C01566=1087.929,-11.575,444.144,174.719,17.924,152.855
C01567=1087.934,-11.325,444.130,174.720,17.925,152.855
C01568=1087.940,-11.076,444.117,174.722,17.927,152.855
C01569=1087.945,-10.826,444.104,174.723,17.928,152.855
C01570=1087.952,-10.577,444.090,174.725,17.930,152.855
C01571=1087.957,-10.327,444.076,174.727,17.932,152.855
C01572=1087.963,-10.077,444.064,174.728,17.934,152.855
C01573=1087.968,-9.828,444.050,174.729,17.935,152.855
C01574=1087.975,-9.578,444.037,174.732,17.937,152.855
C01575=1087.981,-9.329,444.024,174.733,17.939,152.855
C01576=1087.986,-9.079,444.010,174.734,17.940,152.856
C01577=1087.992,-8.830,443.997,174.736,17.942,152.856
C01578=1087.998,-8.580,443.983,174.738,17.944,152.855
C01579=1088.004,-8.331,443.970,174.740,17.945,152.855
C01580=1088.010,-8.081,443.956,174.741,17.947,152.856
C01581=1088.016,-7.831,443.943,174.743,17.948,152.856
C01582=1088.021,-7.581,443.929,174.745,17.950,152.856
C01583=1088.028,-7.332,443.916,174.746,17.952,152.856
C01584=1088.033,-7.082,443.902,174.748,17.954,152.856
C01585=1088.039,-6.833,443.889,174.749,17.955,152.856
C01586=1088.045,-6.583,443.875,174.751,17.957,152.856
C01587=1088.051,-6.334,443.862,174.753,17.959,152.856
C01588=1088.056,-6.084,443.849,174.754,17.960,152.856
C01589=1088.062,-5.835,443.835,174.755,17.962,152.856
C01590=1088.068,-5.585,443.821,174.757,17.964,152.856
C01591=1088.075,-5.335,443.808,174.759,17.966,152.856
C01592=1088.080,-5.086,443.794,174.760,17.967,152.856
C01593=1088.086,-4.836,443.781,174.762,17.969,152.856
C01594=1088.092,-4.587,443.767,174.763,17.970,152.856
C01595=1088.098,-4.338,443.754,174.765,17.973,152.856
C01596=1088.104,-4.088,443.740,174.767,17.974,152.856
C01597=1088.110,-3.839,443.726,174.768,17.976,152.856
C01598=1088.115,-3.589,443.713,174.770,17.977,152.856
C01599=1088.121,-3.339,443.698,174.772,17.979,152.856
C01600=1088.128,-3.090,443.685,174.773,17.981,152.856
C01601=1088.133,-2.840,443.671,174.775,17.982,152.856
C01602=1088.138,-2.590,443.658,174.777,17.985,152.856
C01603=1088.144,-2.341,443.645,174.778,17.986,152.856
C01604=1088.150,-2.091,443.631,174.780,17.988,152.856
C01605=1088.155,-1.841,443.617,174.781,17.989,152.856
C01606=1088.161,-1.592,443.603,174.783,17.991,152.856
C01607=1088.167,-1.343,443.590,174.785,17.993,152.856
C01608=1088.173,-1.069,443.575,174.786,17.995,152.857
C01609=1088.180,-0.794,443.559,174.788,17.997,152.856
C01610=1088.186,-0.521,443.544,174.790,17.998,152.857
C01611=1088.192,-0.247,443.529,174.792,18.000,152.857
C01612=1088.198,0.002,443.515,174.793,18.002,152.857
C01613=1088.203,0.252,443.502,174.795,18.003,152.857
C01614=1088.209,0.501,443.487,174.797,18.006,152.857
C01615=1088.215,0.750,443.473,174.798,18.008,152.857
C01616=1088.221,1.000,443.460,174.799,18.009,152.857
C01617=1088.227,1.250,443.446,174.801,18.011,152.857
C01618=1088.232,1.499,443.432,174.803,18.013,152.857
C01619=1088.238,1.749,443.418,174.804,18.014,152.857
C01620=1088.243,1.999,443.404,174.806,18.016,152.857
C01621=1088.250,2.248,443.391,174.807,18.018,152.857
C01622=1088.255,2.497,443.377,174.809,18.020,152.857
C01623=1088.261,2.748,443.363,174.811,18.021,152.857
C01624=1088.267,2.997,443.348,174.812,18.023,152.857
C01625=1088.272,3.246,443.334,174.814,18.025,152.857
C01626=1088.279,3.496,443.321,174.816,18.027,152.857
C01627=1088.284,3.745,443.307,174.817,18.028,152.857
C01628=1088.290,3.995,443.293,174.819,18.030,152.857
C01629=1088.296,4.245,443.279,174.821,18.032,152.857
C01630=1088.301,4.494,443.264,174.822,18.033,152.857
C01631=1088.307,4.743,443.251,174.824,18.035,152.857
C01632=1088.313,4.993,443.237,174.826,18.037,152.857
C01633=1088.319,5.242,443.223,174.827,18.039,152.857
C01634=1088.325,5.493,443.209,174.829,18.040,152.858
C01635=1088.331,5.742,443.195,174.830,18.042,152.858
C01636=1088.336,5.991,443.181,174.832,18.044,152.858
C01637=1088.341,6.241,443.167,174.834,18.045,152.858
C01638=1088.348,6.491,443.153,174.835,18.047,152.858
C01639=1088.354,6.740,443.139,174.837,18.049,152.858
C01640=1088.360,6.989,443.125,174.839,18.050,152.858
C01641=1088.365,7.239,443.111,174.840,18.052,152.858
C01642=1088.371,7.489,443.097,174.842,18.053,152.858
C01643=1088.377,7.738,443.082,174.844,18.055,152.858
C01644=1088.382,7.988,443.068,174.845,18.057,152.858
C01645=1088.388,8.237,443.054,174.847,18.058,152.858
C01646=1088.395,8.486,443.040,174.849,18.061,152.858
C01647=1088.400,8.736,443.026,174.850,18.062,152.858
C01648=1088.406,8.986,443.012,174.852,18.064,152.858
C01649=1088.412,9.235,442.997,174.853,18.065,152.858
C01650=1088.418,9.485,442.984,174.855,18.067,152.858
C01651=1088.423,9.734,442.970,174.857,18.069,152.858
C01652=1088.429,9.983,442.955,174.858,18.071,152.858
C01653=1088.435,10.234,442.941,174.860,18.073,152.858
C01654=1088.441,10.483,442.927,174.862,18.074,152.858
C01655=1088.446,10.732,442.912,174.863,18.076,152.858
C01656=1088.453,10.982,442.899,174.865,18.078,152.858
C01657=1088.459,11.231,442.884,174.867,18.079,152.858
C01658=1088.464,11.481,442.870,174.868,18.081,152.858
C01659=1088.471,11.731,442.856,174.870,18.082,152.858
C01660=1088.476,11.980,442.842,174.872,18.084,152.858
C01661=1088.482,12.230,442.828,174.874,18.086,152.858
C01662=1088.488,12.479,442.813,174.875,18.087,152.858
C01663=1088.494,12.729,442.799,174.877,18.089,152.858
C01664=1088.499,12.978,442.784,174.879,18.091,152.858
C01665=1088.505,13.228,442.770,174.880,18.093,152.858
C01666=1088.511,13.477,442.755,174.882,18.095,152.858
C01667=1088.517,13.727,442.741,174.884,18.096,152.858
C01668=1088.523,13.976,442.727,174.885,18.098,152.858
C01669=1088.529,14.226,442.713,174.886,18.099,152.858
C01670=1088.535,14.475,442.698,174.889,18.101,152.858
C01671=1088.540,14.725,442.684,174.890,18.103,152.858
C01672=1088.547,15.001,442.668,174.892,18.105,152.858
C01673=1088.554,15.276,442.652,174.894,18.107,152.859
C01674=1088.560,15.552,442.636,174.896,18.109,152.859
C01675=1088.566,15.828,442.621,174.897,18.110,152.859
C01676=1088.572,16.077,442.606,174.899,18.112,152.859
C01677=1088.578,16.327,442.592,174.901,18.114,152.859
C01678=1088.583,16.577,442.577,174.902,18.116,152.859
C01679=1088.589,16.826,442.562,174.905,18.118,152.859
C01680=1088.594,17.075,442.548,174.906,18.119,152.859
C01681=1088.601,17.325,442.533,174.907,18.121,152.859
C01682=1088.606,17.575,442.519,174.910,18.122,152.859
C01683=1088.612,17.823,442.505,174.911,18.124,152.859
C01684=1088.618,18.073,442.490,174.913,18.126,152.859
C01685=1088.623,18.323,442.475,174.915,18.128,152.859
C01686=1088.630,18.573,442.460,174.916,18.129,152.859
C01687=1088.635,18.822,442.447,174.918,18.131,152.859
C01688=1088.641,19.071,442.432,174.920,18.133,152.859
C01689=1088.647,19.321,442.417,174.921,18.134,152.859
C01690=1088.653,19.570,442.403,174.923,18.136,152.859
C01691=1088.658,19.820,442.388,174.925,18.138,152.859
C01692=1088.664,20.069,442.373,174.926,18.140,152.859
C01693=1088.670,20.319,442.359,174.928,18.141,152.859
C01694=1088.676,20.569,442.344,174.930,18.143,152.859
C01695=1088.682,20.818,442.330,174.931,18.145,152.859
C01696=1088.687,21.068,442.315,174.933,18.146,152.859
C01697=1088.693,21.317,442.300,174.935,18.149,152.859
C01698=1088.699,21.566,442.286,174.937,18.150,152.859
C01699=1088.704,21.816,442.270,174.938,18.151,152.859
C01700=1088.710,22.066,442.256,174.940,18.153,152.859
C01701=1088.716,22.315,442.241,174.942,18.155,152.859
C01702=1088.722,22.564,442.227,174.943,18.156,152.859
C01703=1088.728,22.814,442.211,174.945,18.159,152.859
C01704=1088.733,23.064,442.197,174.947,18.160,152.859
C01705=1088.739,23.313,442.183,174.948,18.162,152.859
C01706=1088.744,23.563,442.167,174.950,18.164,152.859
C01707=1088.750,23.812,442.153,174.952,18.165,152.859
C01708=1088.756,24.062,442.138,174.953,18.167,152.859
C01709=1088.762,24.311,442.124,174.955,18.169,152.859
C01710=1088.768,24.561,442.108,174.957,18.171,152.859
C01711=1088.774,24.810,442.094,174.958,18.172,152.859
C01712=1088.780,25.059,442.079,174.961,18.174,152.859
C01713=1088.785,25.309,442.064,174.962,18.175,152.859
C01714=1088.791,25.559,442.049,174.963,18.177,152.859
C01715=1088.797,25.808,442.035,174.966,18.179,152.859
C01716=1088.802,26.058,442.019,174.967,18.181,152.859
C01717=1088.808,26.307,442.005,174.968,18.182,152.860
C01718=1088.815,26.557,441.990,174.971,18.184,152.860
C01719=1088.820,26.806,441.975,174.972,18.186,152.860
C01720=1088.826,27.055,441.960,174.975,18.187,152.859
C01721=1088.832,27.305,441.946,174.976,18.189,152.860
C01722=1088.837,27.555,441.930,174.977,18.190,152.860
C01723=1088.843,27.804,441.916,174.980,18.193,152.860
C01724=1088.849,28.054,441.900,174.981,18.194,152.860
C01725=1088.854,28.303,441.885,174.982,18.196,152.860
C01726=1088.861,28.553,441.871,174.985,18.198,152.860
C01727=1088.866,28.802,441.855,174.986,18.199,152.860
C01728=1088.872,29.051,441.840,174.988,18.200,152.860
C01729=1088.877,29.301,441.825,174.990,18.203,152.860
C01730=1088.884,29.550,441.810,174.991,18.204,152.860
C01731=1088.889,29.800,441.795,174.993,18.206,152.860
C01732=1088.895,30.049,441.780,174.995,18.208,152.860
C01733=1088.900,30.299,441.765,174.996,18.209,152.860
C01734=1088.907,30.548,441.750,174.999,18.211,152.860
C01735=1088.912,30.797,441.735,175.000,18.213,152.860
C01736=1088.918,31.075,441.718,175.002,18.215,152.860
C01737=1088.925,31.352,441.702,175.004,18.217,152.860
C01738=1088.931,31.629,441.685,175.006,18.219,152.860
C01739=1088.937,31.906,441.668,175.007,18.220,152.860
C01740=1088.943,32.156,441.652,175.010,18.222,152.860
C01741=1088.949,32.405,441.638,175.011,18.223,152.860
C01742=1088.954,32.655,441.622,175.013,18.226,152.860
C01743=1088.960,32.904,441.608,175.015,18.227,152.860
C01744=1088.966,33.154,441.592,175.016,18.229,152.860
C01745=1088.971,33.403,441.578,175.018,18.231,152.860
C01746=1088.977,33.653,441.562,175.020,18.232,152.860
C01747=1088.984,33.902,441.546,175.021,18.234,152.860
C01748=1088.989,34.151,441.531,175.024,18.235,152.860
C01749=1088.994,34.401,441.516,175.025,18.237,152.860
C01750=1089.000,34.650,441.501,175.027,18.239,152.860
C01751=1089.006,34.900,441.486,175.029,18.241,152.860
C01752=1089.012,35.150,441.471,175.030,18.242,152.860
C01753=1089.017,35.399,441.455,175.032,18.244,152.860
C01754=1089.024,35.648,441.440,175.034,18.245,152.860
C01755=1089.029,35.897,441.425,175.036,18.248,152.860
C01756=1089.035,36.147,441.409,175.038,18.249,152.860
C01757=1089.041,36.397,441.394,175.039,18.251,152.860
C01758=1089.046,36.646,441.379,175.041,18.253,152.860
C01759=1089.052,36.896,441.364,175.043,18.254,152.860
C01760=1089.058,37.145,441.348,175.044,18.255,152.860
C01761=1089.063,37.395,441.333,175.047,18.257,152.860
C01762=1089.070,37.644,441.318,175.048,18.259,152.860
C01763=1089.075,37.894,441.302,175.050,18.261,152.860
C01764=1089.082,38.143,441.287,175.052,18.262,152.860
C01765=1089.087,38.393,441.271,175.053,18.264,152.860
C01766=1089.092,38.642,441.256,175.056,18.266,152.860
C01767=1089.098,38.892,441.241,175.057,18.267,152.860
C01768=1089.105,39.141,441.225,175.059,18.269,152.860
C01769=1089.110,39.390,441.210,175.061,18.271,152.860
C01770=1089.115,39.640,441.194,175.062,18.272,152.860
C01771=1089.120,39.889,441.179,175.065,18.274,152.860
C01772=1089.126,40.139,441.163,175.066,18.276,152.860
C01773=1089.133,40.388,441.148,175.068,18.278,152.860
C01774=1089.138,40.638,441.133,175.070,18.279,152.860
C01775=1089.144,40.887,441.116,175.071,18.281,152.860
C01776=1089.149,41.137,441.101,175.073,18.283,152.860
C01777=1089.155,41.386,441.086,175.075,18.284,152.860
C01778=1089.161,41.635,441.070,175.077,18.286,152.860
C01779=1089.167,41.885,441.054,175.079,18.288,152.860
C01780=1089.172,42.134,441.039,175.080,18.289,152.860
C01781=1089.178,42.384,441.023,175.082,18.291,152.860
C01782=1089.184,42.633,441.008,175.084,18.292,152.860
C01783=1089.189,42.882,440.992,175.086,18.295,152.860
C01784=1089.195,43.132,440.977,175.087,18.296,152.860
C01785=1089.201,43.382,440.961,175.090,18.298,152.860
C01786=1089.207,43.631,440.945,175.091,18.299,152.860
C01787=1089.212,43.880,440.930,175.093,18.301,152.860
C01788=1089.218,44.130,440.914,175.095,18.303,152.860
C01789=1089.224,44.380,440.898,175.096,18.305,152.860
C01790=1089.229,44.628,440.883,175.099,18.306,152.860
C01791=1089.235,44.878,440.867,175.100,18.308,152.860
C01792=1089.241,45.128,440.851,175.102,18.309,152.860
C01793=1089.246,45.377,440.836,175.104,18.311,152.860
C01794=1089.252,45.627,440.820,175.105,18.313,152.860
C01795=1089.258,45.876,440.804,175.108,18.315,152.860
C01796=1089.263,46.125,440.789,175.109,18.316,152.860
C01797=1089.269,46.375,440.772,175.111,18.318,152.860
C01798=1089.274,46.625,440.757,175.113,18.320,152.860
C01799=1089.280,46.873,440.741,175.114,18.321,152.860
C01800=1089.286,47.151,440.722,175.117,18.323,152.860
C01801=1089.292,47.428,440.706,175.119,18.325,152.860
C01802=1089.299,47.705,440.688,175.121,18.327,152.860
C01803=1089.304,47.983,440.670,175.123,18.329,152.860
C01804=1089.310,48.232,440.654,175.125,18.331,152.860
C01805=1089.316,48.482,440.639,175.126,18.332,152.860
C01806=1089.321,48.731,440.623,175.129,18.334,152.860
C01807=1089.327,48.980,440.606,175.130,18.335,152.860
C01808=1089.333,49.230,440.591,175.132,18.337,152.860
C01809=1089.339,49.479,440.575,175.134,18.339,152.860
C01810=1089.344,49.728,440.559,175.136,18.340,152.860
C01811=1089.350,49.978,440.543,175.138,18.342,152.860
C01812=1089.356,50.227,440.527,175.139,18.344,152.860
C01813=1089.361,50.477,440.511,175.141,18.346,152.860
C01814=1089.367,50.726,440.496,175.143,18.347,152.860
C01815=1089.373,50.975,440.479,175.144,18.348,152.860
C01816=1089.378,51.225,440.464,175.147,18.351,152.860
C01817=1089.384,51.474,440.447,175.148,18.352,152.860
C01818=1089.390,51.724,440.431,175.151,18.354,152.860
C01819=1089.395,51.973,440.416,175.152,18.355,152.860
